// TwinCAT 3 PLC project Plc_Prog
// ProgramVersion: 3.1.4024.0
// libraries:
//   CPNTeck - OSCAT BASIC, * (CPNTeck - Automação Industrial)
//   Tc2_EtherCAT, * (Beckhoff Automation GmbH)
//   Tc2_Standard, * (Beckhoff Automation GmbH)
//   Tc2_SUPS, * (Beckhoff Automation GmbH)
//   Tc2_System, * (Beckhoff Automation GmbH)
//   Tc2_Utilities, * (Beckhoff Automation GmbH)
//   Tc3_Module, * (Beckhoff Automation GmbH)
// project tree:
//   Function Blocks/DELTA - MS300/ C2000_ANALOG_INPUTS.TcDUT (not stored), C2000_ANALOG_OUTPUTS.TcDUT (not stored), C2000_CONTROLWORD.TcDUT (not stored), C2000_DEV_CONFIG.TcDUT, C2000_DIGITAL_INPUTS.TcDUT, C2000_DIGITAL_OUTPUTS.TcDUT (not stored), C2000_DRVTOPLC_PDOS.TcDUT (not stored), C2000_PDOS.TcDUT, C2000_PLCTODRV_PDOS.TcDUT (not stored), C2000_STATUSWORD.TcDUT (not stored), E_C2000_ModeOfOperation.TcDUT, FB_DELTA_C2000_ETC.TcPOU
//   Function Blocks/IOs/Beckhoff/Common/ FB_SavePersistentData.TcPOU (not stored)
//   Function Blocks/IOs/Beckhoff/EL1809 - Digital Inputs/DataTypes/ EL1809_DEV_CONFIG.TcDUT, EL1809_HWTOPLC_PDOS.TcDUT (not stored), EL1809_PDOS.TcDUT
//   Function Blocks/IOs/Beckhoff/EL1809 - Digital Inputs/ FB_EL1809.TcPOU
//   Function Blocks/IOs/Beckhoff/EL3052 - Ai 2 x 4-20MA - 12bit/DataTypes/ EL3052_DEV_CONFIG.TcDUT (not stored), EL3052_DEV_STATUS.TcDUT (not stored), EL3052_HWTOPLC_PDOS.TcDUT (not stored), EL3052_CHANNEL.TcDUT, EL3052_PDOS.TcDUT
//   Function Blocks/IOs/Beckhoff/EL3052 - Ai 2 x 4-20MA - 12bit/ FB_EL3052.TcPOU (not stored)
//   Function Blocks/IOs/Beckhoff/EL2809 - Digital Outputs/DataTypes/ EL2809_DEV_CONFIG.TcDUT (not stored), EL2809_PDOS.TcDUT, EL2809_PLCTOHW_PDOS.TcDUT (not stored)
//   Function Blocks/IOs/Beckhoff/EL2809 - Digital Outputs/ FB_EL2809.TcPOU
//   Function Blocks/IOs/Beckhoff/EL3152 - Ai 2 x 4-20MA - 16bit/DataTypes/ EL3152_CHANNEL.TcDUT (not stored), EL3152_DEV_CONFIG.TcDUT (not stored), EL3152_DEV_STATUS.TcDUT (not stored), EL3152_HWTOPLC_PDOS.TcDUT, EL3152_PDOS.TcDUT (not stored)
//   Function Blocks/IOs/Beckhoff/EL3152 - Ai 2 x 4-20MA - 16bit/ FB_EL3152.TcPOU
//   Function Blocks/IOs/Beckhoff/EL3154 - Ai 4 x 4-20MA - 16bit/DataTypes/ EL3154_CHANNEL.TcDUT, EL3154_DEV_CONFIG.TcDUT (not stored), EL3154_DEV_STATUS.TcDUT (not stored), EL3154_HWTOPLC_PDOS.TcDUT, EL3154_PDOS.TcDUT (not stored)
//   Function Blocks/IOs/Beckhoff/EL3154 - Ai 4 x 4-20MA - 16bit/ FB_EL3154.TcPOU (not stored)
//   Function Blocks/IOs/Beckhoff/EL3204 - Ai 4 x PT100 %28RTD%29/DataTypes/ EL3204_DEV_CONFIG.TcDUT (not stored), EL3204_CHANNEL.TcDUT (not stored), EL3204_DEV_STATUS.TcDUT (not stored), EL3204_HWTOPLC_PDOS.TcDUT (not stored), EL3204_PDOS.TcDUT (not stored)
//   Function Blocks/IOs/Beckhoff/EL3204 - Ai 4 x PT100 %28RTD%29/ FB_EL3204.TcPOU (not stored)
//   Function Blocks/IOs/Beckhoff/EL4024 - AQ 4 x 4-20MA/DataTypes/ EL4024_DEV_CONFIG.TcDUT (not stored), EL4024_HWTOPLC_PDOS.TcDUT (not stored), EL4024_PDOS.TcDUT (not stored)
//   Function Blocks/IOs/Beckhoff/EL4024 - AQ 4 x 4-20MA/ FB_EL4024.TcPOU (not stored)
//   Function Blocks/IOs/Beckhoff/EL6910 - TwinSAFE PLC/ EL6910_ESTOP.TcDUT (not stored), EL6910_ESTOP_DIGNOSTICS.TcDUT (not stored), EL6910_ESTOP_STATUS.TcDUT, EL6910_HWTOPLC_PDOS.TcDUT (not stored), EL6910_PDOS.TcDUT, EL6910_PLCTOHW_PDOS.TcDUT, FB_EL6910.TcPOU (not stored)
//   Function Blocks/PaperMachine/Auxiliary/ FB_FormingBoardDriveControl.TcPOU, FB_FormingBoardRollUpDown.TcPOU, FB_FormingBoardWireStretchControl.TcPOU (not stored), FB_Gen_SRamp.TcPOU (not stored), FB_HeadboxLipsPWMControl.TcPOU (not stored), FB_LevelControl.TcPOU, FB_LevelControl_V2.TcPOU (not stored), FB_MixPumpControl.TcPOU, FB_MixPumpControl_V1.TcPOU, FB_PaperMachine.TcPOU, FB_PressureControl.TcPOU (not stored), FB_PressureControl_V1.TcPOU, FB_VfdProcessControler.TcPOU, FB_ValveProcessControler.TcPOU, FB_SimpleMotorStart.TcPOU, FB_SimpleMotorStart_V2.TcPOU, FB_SimpleMotorStart_V3.TcPOU, FB_SoftstarterSimple.TcPOU (not stored), FB_SoftstarterWithBypass.TcPOU, FB_SoftstarterWithBypass_V1.TcPOU, FB_SpeedDroopControl.TcPOU, FB_SpeedDroopControl_1.TcPOU, FB_WirePitControl.TcPOU, FB_WirePitControl_1.TcPOU (not stored)
//   Function Blocks/PaperMachine/DataTypes/ PaperMachine_TypeHmiConfig.TcDUT, PaperMachine_TypeHmiCommands.TcDUT, PaperMachine_TypeHmiStatus.TcDUT, PaperMachine_TypeHmiAlarms.TcDUT
//   Function Blocks/PaperMachine/DriveControl/ FB_DryingSectionDriveControl_V1.TcPOU (not stored), FB_DryingSectionDriveControl_V2.TcPOU (not stored), FB_DryingSectionDriveControl_V3.TcPOU, FB_FormingBoardControl_V3.TcPOU, FB_PressSectionDriveControl_V2_bak.TcPOU, FB_WinderDriveControl_V1.TcPOU, FB_DryingSectionLubrificationControl_V1.TcPOU, FB_DryingSectionPressureControl.TcPOU (not stored), FB_FormingBoardControl_V1.TcPOU, FB_PressSectionDriveControl_V1.TcPOU (not stored), FB_PressSectionDriveControl_V2.TcPOU
//   Function Blocks/PaperMachine/ FB_AlarmControl.TcPOU, FB_GroupDisplayFilters_V1.TcPOU, FB_GroupDriveControl_V1.TcPOU (not stored), FB_GroupSpeedControl_V1.TcPOU, FB_FormingBoardSpeedControl.TcPOU, FB_DryingSecSpeedControl.TcPOU, FB_WinderSpeedControl.TcPOU, FB_GroupTorqueTrimControl_V1.TcPOU, FB_GroupTorqueTrimControl_V2.TcPOU
//   Function Blocks/Rewinder/DataTypes/ RewinderConfig_TypeStruct.TcDUT (not stored), Rewinder_TypePressRoll.TcDUT, Rewinder_TypeBrakeControl.TcDUT
//   Function Blocks/Rewinder/ FB_RewinderControl_V1.TcPOU (not stored)
//   GVLs/ GVL_Hw.TcGVL (not stored)
//   / PlcTask.TcTTO
//   POUs/Implicit Checks/ CheckBounds.TcPOU (not stored), CheckDivDInt.TcPOU, CheckDivLInt.TcPOU, CheckDivLReal.TcPOU (not stored), CheckDivReal.TcPOU (not stored), CheckLRangeSigned.TcPOU (not stored), CheckLRangeUnsigned.TcPOU (not stored), CheckPointer.TcPOU (not stored), CheckRangeSigned.TcPOU (not stored), CheckRangeUnsigned.TcPOU
//   POUs/ MAIN.TcPOU
// real-time tasks:
//   TASK PlcTask: cycle T#5ms, priority 20, ADS port 350
// I/O:
//   DEVICE ETH, AmsNetId 192.168.100.1.3.1
//     +P5=050-BC1 - PLC Cabinet [EK1100 EtherCAT Coupler (2A E-Bus)]
//       +P5=050-DI1 (EL1809) [EL1809 16Ch. Dig. Input 24V, 3ms]
//       +P5=050-DI2 (EL1809) [EL1809 16Ch. Dig. Input 24V, 3ms]
//       +P5=050-DI3 (EL1809) [EL1809 16Ch. Dig. Input 24V, 3ms]
//       +P5=050-DO1 (EL2809) [EL2809 16Ch. Dig. Output 24V, 0.5A]
//       +P5=050-DO2 (EL2809) [EL2809 16Ch. Dig. Output 24V, 0.5A]
//       +P5=050-DO3 (EL2809) [EL2809 16Ch. Dig. Output 24V, 0.5A]
//       +P5=050-SP1 (EL6910) [EL6910, TwinSAFE PLC]
//       +P5=050-SI1 (EL1918) [EL1918, 8Ch. Safety Input 24V, TwinSAFE]
//         modules: Module 1 (FSOE), Module 2 (FSLOGIC)
//       +P5=050-SO1 (EL2904) [EL2904, 4 Ch. Safety Output 24V, 0.5A, TwinSAFE]
//         modules: Module 1 (FSOES), Module 2 (DO)
//       +P5=050-SO2 (EL2904) [EL2904, 4 Ch. Safety Output 24V, 0.5A, TwinSAFE]
//         modules: Module 1 (FSOES), Module 2 (DO)
//       +P5=050-BC2 [EL6601 1 Port Switch (Ethernet, CoE)]
//       +P5=050-BC3 [EL6601 1 Port Switch (Ethernet, CoE)]
//       +P5=050-BE1 [EL9011 End Terminal]
//     +P5=050-BC2 - PLC Cabinet [EK1100 EtherCAT Coupler (2A E-Bus)]
//       +P5=050-AI (EL3052) [EL3052 2Ch. Ana. Input 4-20mA]
//       +P5=050-AI2 (EL3152) [EL3152 2Ch. Ana Input 4-20mA]
//       +P5=050-AI3 (EL3052) [EL3052 2Ch. Ana. Input 4-20mA]
//       +P5=050-AI4 (EL3052) [EL3052 2Ch. Ana. Input 4-20mA]
//       +P5=050-BE2 [EL9011 End Terminal]
//     +P4=300-UG1 - Mix Pump [Delta CH2000 EtherCAT(CoE)]
//     +P3=300-UG1 - WirePit Pump [Delta CH2000 EtherCAT(CoE)]
//     +P3=100-UG1 - SuctionRoll [Delta CH2000 EtherCAT(CoE)]
//     +P3=100-UG1 - CouchPit [Delta CH2000 EtherCAT(CoE)]
//     +P3=100-UG2 - Stock pump [Delta CH2000 EtherCAT(CoE)]
//     +P2=100-UG1 - Drive Roll [Delta CH2000 EtherCAT(CoE)]
//     +P9=050-BC1 - Vaccum PLC Cabinet [EK1100 EtherCAT Coupler (2A E-Bus)]
//       +P9=050-DI1 (EL1809) [EL1809 16Ch. Dig. Input 24V, 3ms]
//       +P9=050-DI2 (EL1809) [EL1809 16Ch. Dig. Input 24V, 3ms]
//       +P9=050-DI3 (EL1809) [EL1809 16Ch. Dig. Input 24V, 3ms]
//       +P9=050-DO1 (EL2809) [EL2809 16Ch. Dig. Output 24V, 0.5A]
//       +P9=050-DO2 (EL2809) [EL2809 16Ch. Dig. Output 24V, 0.5A]
//       +P9=050-DO3 (EL2809) [EL2809 16Ch. Dig. Output 24V, 0.5A]
//       +P9=050-AI1 (EL3054) [EL3054 4Ch. Ana. Input 4-20mA]
//       Term 101 (EL3052) [EL3052 2Ch. Ana. Input 4-20mA]
//       Term 102 (EL4004) [EL4004 4Ch. Ana. Output 0-10V, 12bit]
//       Term 151 (EL9011) [EL9011 End Terminal]
//       +P9=050-BE1 [EL9011 End Terminal]
//     +P10=050-BC1 - Press / Dryer PLC Cabinet [EK1100 EtherCAT Coupler (2A E-Bus)]
//       +P10=050-DI1 (EL1809) [EL1809 16Ch. Dig. Input 24V, 3ms]
//       +P10=050-DI2 (EL1809) [EL1809 16Ch. Dig. Input 24V, 3ms]
//       +P10=050-DI3 (EL1809) [EL1809 16Ch. Dig. Input 24V, 3ms]
//       +P10=050-DI4 (EL1809) [EL1809 16Ch. Dig. Input 24V, 3ms]
//       +P10=050-DI5 (EL1809) [EL1809 16Ch. Dig. Input 24V, 3ms]
//       +P10=050-DI6 (EL1809) [EL1809 16Ch. Dig. Input 24V, 3ms]
//       +P10=050-DI7 (EL1809) [EL1809 16Ch. Dig. Input 24V, 3ms]
//       +P10=050-DI8 (EL1809) [EL1809 16Ch. Dig. Input 24V, 3ms]
//       +P10=050-DO1 (EL2809) [EL2809 16Ch. Dig. Output 24V, 0.5A]
//       +P10=050-DO2 (EL2809) [EL2809 16Ch. Dig. Output 24V, 0.5A]
//       +P10=050-DO3 (EL2809) [EL2809 16Ch. Dig. Output 24V, 0.5A]
//       +P10=050-DO4 (EL2809) [EL2809 16Ch. Dig. Output 24V, 0.5A]
//       +P10=050-SI1 (EL1918) [EL1918, 8Ch. Safety Input 24V, TwinSAFE]
//         modules: Module 1 (FSOE), Module 2 (FSLOGIC)
//       +P10=050-SO1 (EL2904) [EL2904, 4 Ch. Safety Output 24V, 0.5A, TwinSAFE]
//         modules: Module 1 (FSOES), Module 2 (DO)
//       +P10=050-BE1 [EL9011 End Terminal]
//     +P10=050-BC2 - Press / Dryer PLC Cabinet [EK1100 EtherCAT Coupler (2A E-Bus)]
//       +P10=050-AI1 (EL3054) [EL3054 4Ch. Ana. Input 4-20mA]
//       +P10=050-AI2 (EL3204) [EL3204 4Ch. Ana. Input PT100 (RTD)]
//       +P10=050-AO1(EL4024) [EL4024 4Ch. Ana. Output 4-20mA, 12bit]
//       +P10=050-BE2 [EL9011 End Terminal]
//     +P11=400-UG1 - Second Press [Delta C2000Plus EtherCAT(CoE)]
//     +P12=400-UG1 - First Press [Delta C2000Plus EtherCAT(CoE)]
//     +P13=500-UG1 - Dryer Section GR1 - Upper GR1 Slave [Delta C2000Plus EtherCAT(CoE)]
//     +P12=500-UG2 - Dryer Section GR1 - Lower GR1 Master [Delta C2000Plus EtherCAT(CoE)]
//     +P12=500-UG3 - Dryer Section GR1 - Upper Master [Delta CH2000 EtherCAT(CoE)]
//     +P12=501-UG1 - Dryer Section  GR2 - Lower Slave [Delta C2000Plus EtherCAT(CoE)]
//     +P12=501-UG2 - Dryer Section GR2 - Upper Slave [Delta CH2000 EtherCAT(CoE)]
//     +P12=501-UG3 - Dryer Section GR2 - Lower Master [Delta C2000Plus EtherCAT(CoE)]
//     +P13=501-UG1 - Dryer Section GR2 - Upper Master [Delta CH2000 EtherCAT(CoE)]
//     +P13=502-UG2 - Dryer Section GR3 - Lower Slave [Delta C2000Plus EtherCAT(CoE)]
//     +P13=502-UG2 - Dryer Section GR3 - Upper Slave [Delta C2000Plus EtherCAT(CoE)]
//     +P13=502-UG3 - Dryer Section GR3 - Lower Master [Delta C2000Plus EtherCAT(CoE)]
//     +P13=502-UG4 - Dryer Section GR3 - Upper Master [Delta C2000Plus EtherCAT(CoE)]
//     +P14=600-UG1 - Winder [Delta C2000Plus EtherCAT(CoE)]
//     +CP2=050-BC1 - Winder command panel [EK1100 EtherCAT Coupler (2A E-Bus)]
//       +CP2=050-SI1 (EL1918) [EL1918, 8Ch. Safety Input 24V, TwinSAFE]
//         modules: Module 1 (FSOE), Module 2 (FSLOGIC)
//       +CP2=050-DI1 (EL1809) [EL1809 16Ch. Dig. Input 24V, 3ms]
//       +CP2=050-DO1 (EL2809 [EL2809 16Ch. Dig. Output 24V, 0.5A]
//       +CP2=050-AO1 (EL4024) [EL4024 4Ch. Ana. Output 4-20mA, 12bit]
//       +CP2=050-BE1 (EL4024) [EL9011 End Terminal]
// variable links:
//   ETH <-> ETH/+CP2=050-BC1 - Winder command panel/+CP2=050-SI1 (EL1918)
//     +P5=050-BC1 - PLC Cabinet/+P5=050-SP1 (EL6910)/ConnectionInputs/TwinSafeGroup1.+CP2=050-SI1 (EL1918) - Module 1 (FSOE)_9 TxPDO <-> Module 1 (FSOE)/FSoE Outputs/FSOE
//     +P5=050-BC1 - PLC Cabinet/+P5=050-SP1 (EL6910)/ConnectionOutputs/TwinSafeGroup1.+CP2=050-SI1 (EL1918) - Module 1 (FSOE)_9 RxPDO <-> Module 1 (FSOE)/FSoE Inputs/FSOE
//   ETH <-> ETH/+P10=050-BC1 - Press / Dryer PLC Cabinet/+P10=050-SI1 (EL1918)
//     +P5=050-BC1 - PLC Cabinet/+P5=050-SP1 (EL6910)/ConnectionInputs/TwinSafeGroup1.+P10=050-SI1 (EL1918) - Module 1 (FSOE)_7 TxPDO <-> Module 1 (FSOE)/FSoE Outputs/FSOE
//   ETH <-> ETH/+P10=050-BC1 - Press / Dryer PLC Cabinet/+P10=050-SO1 (EL2904)
//     +P5=050-BC1 - PLC Cabinet/+P5=050-SP1 (EL6910)/ConnectionInputs/TwinSafeGroup1.+P10=050-SO1 (EL2904) - Module 1 (FSOES)_8 TxPDO <-> Module 1 (FSOES)/RxPDO/FSOE
//     +P5=050-BC1 - PLC Cabinet/+P5=050-SP1 (EL6910)/ConnectionOutputs/TwinSafeGroup1.+P10=050-SO1 (EL2904) - Module 1 (FSOES)_8 RxPDO <-> Module 1 (FSOES)/TxPDO/FSOE
//   ETH <-> ETH/+P5=050-BC1 - PLC Cabinet/+P5=050-SI1 (EL1918)
//     +P5=050-BC1 - PLC Cabinet/+P5=050-SP1 (EL6910)/ConnectionInputs/TwinSafeGroup1.Term 9 (EL1918) - Module 1 (FSOE)_3 TxPDO <-> Module 1 (FSOE)/FSoE Outputs/FSOE
//   ETH <-> ETH/+P5=050-BC1 - PLC Cabinet/+P5=050-SP1 (EL6910)
//     +P10=050-BC1 - Press / Dryer PLC Cabinet/+P10=050-SI1 (EL1918)/Module 1 (FSOE)/FSoE Inputs/FSOE <-> ConnectionOutputs/TwinSafeGroup1.+P10=050-SI1 (EL1918) - Module 1 (FSOE)_7 RxPDO
//     +P5=050-BC1 - PLC Cabinet/+P5=050-SI1 (EL1918)/Module 1 (FSOE)/FSoE Inputs/FSOE <-> ConnectionOutputs/TwinSafeGroup1.Term 9 (EL1918) - Module 1 (FSOE)_3 RxPDO
//     +P5=050-BC1 - PLC Cabinet/+P5=050-SO1 (EL2904)/Module 1 (FSOES)/RxPDO/FSOE <-> ConnectionInputs/TwinSafeGroup1.Term 10 (EL2904) - Module 1 (FSOES)_4 TxPDO
//     +P5=050-BC1 - PLC Cabinet/+P5=050-SO2 (EL2904)/Module 1 (FSOES)/RxPDO/FSOE <-> ConnectionInputs/TwinSafeGroup1.Term 11 (EL2904) - Module 1 (FSOES)_5 TxPDO
//     +P5=050-BC1 - PLC Cabinet/+P5=050-SO1 (EL2904)/Module 1 (FSOES)/TxPDO/FSOE <-> ConnectionOutputs/TwinSafeGroup1.Term 10 (EL2904) - Module 1 (FSOES)_4 RxPDO
//     +P5=050-BC1 - PLC Cabinet/+P5=050-SO2 (EL2904)/Module 1 (FSOES)/TxPDO/FSOE <-> ConnectionOutputs/TwinSafeGroup1.Term 11 (EL2904) - Module 1 (FSOES)_5 RxPDO
//   Plc_Prog/Plc_Prog Instance <-> ETH/+CP2=050-BC1 - Winder command panel/+CP2=050-AO1 (EL4024)
//     PlcTask Outputs/.CP1_050_AO1.PDOS.HwToPLC.Channel1 <-> AO Outputs Channel 1/Analog output
//     PlcTask Outputs/.CP1_050_AO1.PDOS.HwToPLC.Channel2 <-> AO Outputs Channel 2/Analog output
//     PlcTask Outputs/.CP1_050_AO1.PDOS.HwToPLC.Channel3 <-> AO Outputs Channel 3/Analog output
//     PlcTask Outputs/.CP1_050_AO1.PDOS.HwToPLC.Channel4 <-> AO Outputs Channel 4/Analog output
//   Plc_Prog/Plc_Prog Instance <-> ETH/+CP2=050-BC1 - Winder command panel/+CP2=050-DI1 (EL1809)
//     PlcTask Inputs/.CP1_050_DI1.PDOS.digitalInput_01 <-> Channel 1/Input
//     PlcTask Inputs/.CP1_050_DI1.PDOS.digitalInput_02 <-> Channel 2/Input
//     PlcTask Inputs/.CP1_050_DI1.PDOS.digitalInput_03 <-> Channel 3/Input
//     PlcTask Inputs/.CP1_050_DI1.PDOS.digitalInput_04 <-> Channel 4/Input
//     PlcTask Inputs/.CP1_050_DI1.PDOS.digitalInput_05 <-> Channel 5/Input
//     PlcTask Inputs/.CP1_050_DI1.PDOS.digitalInput_06 <-> Channel 6/Input
//     PlcTask Inputs/.CP1_050_DI1.PDOS.digitalInput_07 <-> Channel 7/Input
//     PlcTask Inputs/.CP1_050_DI1.PDOS.digitalInput_08 <-> Channel 8/Input
//     PlcTask Inputs/.CP1_050_DI1.PDOS.digitalInput_09 <-> Channel 9/Input
//     PlcTask Inputs/.CP1_050_DI1.PDOS.digitalInput_10 <-> Channel 10/Input
//     PlcTask Inputs/.CP1_050_DI1.PDOS.digitalInput_11 <-> Channel 11/Input
//     PlcTask Inputs/.CP1_050_DI1.PDOS.digitalInput_12 <-> Channel 12/Input
//     PlcTask Inputs/.CP1_050_DI1.PDOS.digitalInput_13 <-> Channel 13/Input
//     PlcTask Inputs/.CP1_050_DI1.PDOS.digitalInput_14 <-> Channel 14/Input
//     PlcTask Inputs/.CP1_050_DI1.PDOS.digitalInput_15 <-> Channel 15/Input
//     PlcTask Inputs/.CP1_050_DI1.PDOS.digitalInput_16 <-> Channel 16/Input
//   Plc_Prog/Plc_Prog Instance <-> ETH/+CP2=050-BC1 - Winder command panel/+CP2=050-DO1 (EL2809
//     PlcTask Outputs/.CP1_050_DO1.PDOS.PlcToHw.digitalOutput_01 <-> Channel 1/Output
//     PlcTask Outputs/.CP1_050_DO1.PDOS.PlcToHw.digitalOutput_02 <-> Channel 2/Output
//     PlcTask Outputs/.CP1_050_DO1.PDOS.PlcToHw.digitalOutput_03 <-> Channel 3/Output
//     PlcTask Outputs/.CP1_050_DO1.PDOS.PlcToHw.digitalOutput_04 <-> Channel 4/Output
//     PlcTask Outputs/.CP1_050_DO1.PDOS.PlcToHw.digitalOutput_05 <-> Channel 5/Output
//     PlcTask Outputs/.CP1_050_DO1.PDOS.PlcToHw.digitalOutput_06 <-> Channel 6/Output
//     PlcTask Outputs/.CP1_050_DO1.PDOS.PlcToHw.digitalOutput_07 <-> Channel 7/Output
//     PlcTask Outputs/.CP1_050_DO1.PDOS.PlcToHw.digitalOutput_08 <-> Channel 8/Output
//     PlcTask Outputs/.CP1_050_DO1.PDOS.PlcToHw.digitalOutput_09 <-> Channel 9/Output
//     PlcTask Outputs/.CP1_050_DO1.PDOS.PlcToHw.digitalOutput_10 <-> Channel 10/Output
//     PlcTask Outputs/.CP1_050_DO1.PDOS.PlcToHw.digitalOutput_11 <-> Channel 11/Output
//     PlcTask Outputs/.CP1_050_DO1.PDOS.PlcToHw.digitalOutput_12 <-> Channel 12/Output
//     PlcTask Outputs/.CP1_050_DO1.PDOS.PlcToHw.digitalOutput_13 <-> Channel 13/Output
//     PlcTask Outputs/.CP1_050_DO1.PDOS.PlcToHw.digitalOutput_14 <-> Channel 14/Output
//     PlcTask Outputs/.CP1_050_DO1.PDOS.PlcToHw.digitalOutput_15 <-> Channel 15/Output
//     PlcTask Outputs/.CP1_050_DO1.PDOS.PlcToHw.digitalOutput_16 <-> Channel 16/Output
//   Plc_Prog/Plc_Prog Instance <-> ETH/+P10=050-BC1 - Press / Dryer PLC Cabinet/+P10=050-DI1 (EL1809)
//     PlcTask Inputs/.P10_050_DI1.PDOS.digitalInput_01 <-> Channel 1/Input
//     PlcTask Inputs/.P10_050_DI1.PDOS.digitalInput_02 <-> Channel 2/Input
//     PlcTask Inputs/.P10_050_DI1.PDOS.digitalInput_03 <-> Channel 3/Input
//     PlcTask Inputs/.P10_050_DI1.PDOS.digitalInput_04 <-> Channel 4/Input
//     PlcTask Inputs/.P10_050_DI1.PDOS.digitalInput_05 <-> Channel 5/Input
//     PlcTask Inputs/.P10_050_DI1.PDOS.digitalInput_06 <-> Channel 6/Input
//     PlcTask Inputs/.P10_050_DI1.PDOS.digitalInput_07 <-> Channel 7/Input
//     PlcTask Inputs/.P10_050_DI1.PDOS.digitalInput_08 <-> Channel 8/Input
//     PlcTask Inputs/.P10_050_DI1.PDOS.digitalInput_09 <-> Channel 9/Input
//     PlcTask Inputs/.P10_050_DI1.PDOS.digitalInput_10 <-> Channel 10/Input
//     PlcTask Inputs/.P10_050_DI1.PDOS.digitalInput_11 <-> Channel 11/Input
//     PlcTask Inputs/.P10_050_DI1.PDOS.digitalInput_12 <-> Channel 12/Input
//     PlcTask Inputs/.P10_050_DI1.PDOS.digitalInput_13 <-> Channel 13/Input
//     PlcTask Inputs/.P10_050_DI1.PDOS.digitalInput_14 <-> Channel 14/Input
//     PlcTask Inputs/.P10_050_DI1.PDOS.digitalInput_15 <-> Channel 15/Input
//     PlcTask Inputs/.P10_050_DI1.PDOS.digitalInput_16 <-> Channel 16/Input
//   Plc_Prog/Plc_Prog Instance <-> ETH/+P10=050-BC1 - Press / Dryer PLC Cabinet/+P10=050-DI2 (EL1809)
//     PlcTask Inputs/.P10_050_DI2.PDOS.digitalInput_01 <-> Channel 1/Input
//     PlcTask Inputs/.P10_050_DI2.PDOS.digitalInput_02 <-> Channel 2/Input
//     PlcTask Inputs/.P10_050_DI2.PDOS.digitalInput_03 <-> Channel 3/Input
//     PlcTask Inputs/.P10_050_DI2.PDOS.digitalInput_04 <-> Channel 4/Input
//     PlcTask Inputs/.P10_050_DI2.PDOS.digitalInput_05 <-> Channel 5/Input
//     PlcTask Inputs/.P10_050_DI2.PDOS.digitalInput_06 <-> Channel 6/Input
//     PlcTask Inputs/.P10_050_DI2.PDOS.digitalInput_07 <-> Channel 7/Input
//     PlcTask Inputs/.P10_050_DI2.PDOS.digitalInput_08 <-> Channel 8/Input
//     PlcTask Inputs/.P10_050_DI2.PDOS.digitalInput_09 <-> Channel 9/Input
//     PlcTask Inputs/.P10_050_DI2.PDOS.digitalInput_10 <-> Channel 10/Input
//     PlcTask Inputs/.P10_050_DI2.PDOS.digitalInput_12 <-> Channel 12/Input
//     PlcTask Inputs/.P10_050_DI2.PDOS.digitalInput_13 <-> Channel 13/Input
//     PlcTask Inputs/.P10_050_DI2.PDOS.digitalInput_14 <-> Channel 14/Input
//     PlcTask Inputs/.P10_050_DI2.PDOS.digitalInput_15 <-> Channel 15/Input
//     PlcTask Inputs/.P10_050_DI2.PDOS.digitalInput_16 <-> Channel 16/Input
//     PlcTask Inputs/.P10_050_DI2.PDOS.digitalInput_11 <-> Channel 11/.P10_050_DI2.PDOS.digitalInput_11
//   Plc_Prog/Plc_Prog Instance <-> ETH/+P10=050-BC1 - Press / Dryer PLC Cabinet/+P10=050-DI3 (EL1809)
//     PlcTask Inputs/.P10_050_DI3.PDOS.digitalInput_01 <-> Channel 1/Input
//     PlcTask Inputs/.P10_050_DI3.PDOS.digitalInput_02 <-> Channel 2/Input
//     PlcTask Inputs/.P10_050_DI3.PDOS.digitalInput_03 <-> Channel 3/Input
//     PlcTask Inputs/.P10_050_DI3.PDOS.digitalInput_04 <-> Channel 4/Input
//     PlcTask Inputs/.P10_050_DI3.PDOS.digitalInput_05 <-> Channel 5/Input
//     PlcTask Inputs/.P10_050_DI3.PDOS.digitalInput_06 <-> Channel 6/Input
//     PlcTask Inputs/.P10_050_DI3.PDOS.digitalInput_07 <-> Channel 7/Input
//     PlcTask Inputs/.P10_050_DI3.PDOS.digitalInput_08 <-> Channel 8/Input
//     PlcTask Inputs/.P10_050_DI3.PDOS.digitalInput_09 <-> Channel 9/Input
//     PlcTask Inputs/.P10_050_DI3.PDOS.digitalInput_10 <-> Channel 10/Input
//     PlcTask Inputs/.P10_050_DI3.PDOS.digitalInput_11 <-> Channel 11/Input
//     PlcTask Inputs/.P10_050_DI3.PDOS.digitalInput_12 <-> Channel 12/Input
//     PlcTask Inputs/.P10_050_DI3.PDOS.digitalInput_13 <-> Channel 13/Input
//     PlcTask Inputs/.P10_050_DI3.PDOS.digitalInput_14 <-> Channel 14/Input
//     PlcTask Inputs/.P10_050_DI3.PDOS.digitalInput_15 <-> Channel 15/Input
//     PlcTask Inputs/.P10_050_DI3.PDOS.digitalInput_16 <-> Channel 16/Input
//   Plc_Prog/Plc_Prog Instance <-> ETH/+P10=050-BC1 - Press / Dryer PLC Cabinet/+P10=050-DI4 (EL1809)
//     PlcTask Inputs/.P10_050_DI4.PDOS.digitalInput_01 <-> Channel 1/Input
//     PlcTask Inputs/.P10_050_DI4.PDOS.digitalInput_02 <-> Channel 2/Input
//     PlcTask Inputs/.P10_050_DI4.PDOS.digitalInput_03 <-> Channel 3/Input
//     PlcTask Inputs/.P10_050_DI4.PDOS.digitalInput_04 <-> Channel 4/Input
//     PlcTask Inputs/.P10_050_DI4.PDOS.digitalInput_05 <-> Channel 5/Input
//     PlcTask Inputs/.P10_050_DI4.PDOS.digitalInput_06 <-> Channel 6/Input
//     PlcTask Inputs/.P10_050_DI4.PDOS.digitalInput_07 <-> Channel 7/Input
//     PlcTask Inputs/.P10_050_DI4.PDOS.digitalInput_08 <-> Channel 8/Input
//     PlcTask Inputs/.P10_050_DI4.PDOS.digitalInput_09 <-> Channel 9/Input
//     PlcTask Inputs/.P10_050_DI4.PDOS.digitalInput_10 <-> Channel 10/Input
//     PlcTask Inputs/.P10_050_DI4.PDOS.digitalInput_11 <-> Channel 11/Input
//     PlcTask Inputs/.P10_050_DI4.PDOS.digitalInput_12 <-> Channel 12/Input
//     PlcTask Inputs/.P10_050_DI4.PDOS.digitalInput_13 <-> Channel 13/Input
//     PlcTask Inputs/.P10_050_DI4.PDOS.digitalInput_14 <-> Channel 14/Input
//     PlcTask Inputs/.P10_050_DI4.PDOS.digitalInput_15 <-> Channel 15/Input
//     PlcTask Inputs/.P10_050_DI4.PDOS.digitalInput_16 <-> Channel 16/Input
//   Plc_Prog/Plc_Prog Instance <-> ETH/+P10=050-BC1 - Press / Dryer PLC Cabinet/+P10=050-DI5 (EL1809)
//     PlcTask Inputs/.P10_050_DI5.PDOS.digitalInput_01 <-> Channel 1/Input
//     PlcTask Inputs/.P10_050_DI5.PDOS.digitalInput_02 <-> Channel 2/Input
//     PlcTask Inputs/.P10_050_DI5.PDOS.digitalInput_03 <-> Channel 3/Input
//     PlcTask Inputs/.P10_050_DI5.PDOS.digitalInput_04 <-> Channel 4/Input
//     PlcTask Inputs/.P10_050_DI5.PDOS.digitalInput_05 <-> Channel 5/Input
//     PlcTask Inputs/.P10_050_DI5.PDOS.digitalInput_06 <-> Channel 6/Input
//     PlcTask Inputs/.P10_050_DI5.PDOS.digitalInput_07 <-> Channel 7/Input
//     PlcTask Inputs/.P10_050_DI5.PDOS.digitalInput_08 <-> Channel 8/Input
//     PlcTask Inputs/.P10_050_DI5.PDOS.digitalInput_09 <-> Channel 9/Input
//     PlcTask Inputs/.P10_050_DI5.PDOS.digitalInput_10 <-> Channel 10/Input
//     PlcTask Inputs/.P10_050_DI5.PDOS.digitalInput_11 <-> Channel 11/Input
//     PlcTask Inputs/.P10_050_DI5.PDOS.digitalInput_12 <-> Channel 12/Input
//     PlcTask Inputs/.P10_050_DI5.PDOS.digitalInput_13 <-> Channel 13/Input
//     PlcTask Inputs/.P10_050_DI5.PDOS.digitalInput_14 <-> Channel 14/Input
//     PlcTask Inputs/.P10_050_DI5.PDOS.digitalInput_15 <-> Channel 15/Input
//     PlcTask Inputs/.P10_050_DI5.PDOS.digitalInput_16 <-> Channel 16/Input
//   Plc_Prog/Plc_Prog Instance <-> ETH/+P10=050-BC1 - Press / Dryer PLC Cabinet/+P10=050-DI6 (EL1809)
//     PlcTask Inputs/.P10_050_DI6.PDOS.digitalInput_01 <-> Channel 1/Input
//     PlcTask Inputs/.P10_050_DI6.PDOS.digitalInput_02 <-> Channel 2/Input
//     PlcTask Inputs/.P10_050_DI6.PDOS.digitalInput_03 <-> Channel 3/Input
//     PlcTask Inputs/.P10_050_DI6.PDOS.digitalInput_04 <-> Channel 4/Input
//     PlcTask Inputs/.P10_050_DI6.PDOS.digitalInput_05 <-> Channel 5/Input
//     PlcTask Inputs/.P10_050_DI6.PDOS.digitalInput_06 <-> Channel 6/Input
//     PlcTask Inputs/.P10_050_DI6.PDOS.digitalInput_07 <-> Channel 7/Input
//     PlcTask Inputs/.P10_050_DI6.PDOS.digitalInput_08 <-> Channel 8/Input
//     PlcTask Inputs/.P10_050_DI6.PDOS.digitalInput_09 <-> Channel 9/Input
//     PlcTask Inputs/.P10_050_DI6.PDOS.digitalInput_10 <-> Channel 10/Input
//     PlcTask Inputs/.P10_050_DI6.PDOS.digitalInput_11 <-> Channel 11/Input
//     PlcTask Inputs/.P10_050_DI6.PDOS.digitalInput_12 <-> Channel 12/Input
//     PlcTask Inputs/.P10_050_DI6.PDOS.digitalInput_13 <-> Channel 13/Input
//     PlcTask Inputs/.P10_050_DI6.PDOS.digitalInput_14 <-> Channel 14/Input
//     PlcTask Inputs/.P10_050_DI6.PDOS.digitalInput_15 <-> Channel 15/Input
//     PlcTask Inputs/.P10_050_DI6.PDOS.digitalInput_16 <-> Channel 16/Input
//   Plc_Prog/Plc_Prog Instance <-> ETH/+P10=050-BC1 - Press / Dryer PLC Cabinet/+P10=050-DI7 (EL1809)
//     PlcTask Inputs/.P10_050_DI7.PDOS.digitalInput_01 <-> Channel 1/Input
//     PlcTask Inputs/.P10_050_DI7.PDOS.digitalInput_02 <-> Channel 2/Input
//     PlcTask Inputs/.P10_050_DI7.PDOS.digitalInput_03 <-> Channel 3/Input
//     PlcTask Inputs/.P10_050_DI7.PDOS.digitalInput_04 <-> Channel 4/Input
//     PlcTask Inputs/.P10_050_DI7.PDOS.digitalInput_05 <-> Channel 5/Input
//     PlcTask Inputs/.P10_050_DI7.PDOS.digitalInput_06 <-> Channel 6/Input
//     PlcTask Inputs/.P10_050_DI7.PDOS.digitalInput_07 <-> Channel 7/Input
//     PlcTask Inputs/.P10_050_DI7.PDOS.digitalInput_08 <-> Channel 8/Input
//     PlcTask Inputs/.P10_050_DI7.PDOS.digitalInput_09 <-> Channel 9/Input
//     PlcTask Inputs/.P10_050_DI7.PDOS.digitalInput_10 <-> Channel 10/Input
//     PlcTask Inputs/.P10_050_DI7.PDOS.digitalInput_11 <-> Channel 11/Input
//     PlcTask Inputs/.P10_050_DI7.PDOS.digitalInput_12 <-> Channel 12/Input
//     PlcTask Inputs/.P10_050_DI7.PDOS.digitalInput_13 <-> Channel 13/Input
//     PlcTask Inputs/.P10_050_DI7.PDOS.digitalInput_14 <-> Channel 14/Input
//     PlcTask Inputs/.P10_050_DI7.PDOS.digitalInput_15 <-> Channel 15/Input
//     PlcTask Inputs/.P10_050_DI7.PDOS.digitalInput_16 <-> Channel 16/Input
//   Plc_Prog/Plc_Prog Instance <-> ETH/+P10=050-BC1 - Press / Dryer PLC Cabinet/+P10=050-DI8 (EL1809)
//     PlcTask Inputs/.P10_050_DI8.PDOS.digitalInput_01 <-> Channel 1/Input
//     PlcTask Inputs/.P10_050_DI8.PDOS.digitalInput_02 <-> Channel 2/Input
//     PlcTask Inputs/.P10_050_DI8.PDOS.digitalInput_03 <-> Channel 3/Input
//     PlcTask Inputs/.P10_050_DI8.PDOS.digitalInput_04 <-> Channel 4/Input
//     PlcTask Inputs/.P10_050_DI8.PDOS.digitalInput_05 <-> Channel 5/Input
//     PlcTask Inputs/.P10_050_DI8.PDOS.digitalInput_06 <-> Channel 6/Input
//     PlcTask Inputs/.P10_050_DI8.PDOS.digitalInput_07 <-> Channel 7/Input
//     PlcTask Inputs/.P10_050_DI8.PDOS.digitalInput_08 <-> Channel 8/Input
//     PlcTask Inputs/.P10_050_DI8.PDOS.digitalInput_09 <-> Channel 9/Input
//     PlcTask Inputs/.P10_050_DI8.PDOS.digitalInput_10 <-> Channel 10/Input
//     PlcTask Inputs/.P10_050_DI8.PDOS.digitalInput_11 <-> Channel 11/Input
//     PlcTask Inputs/.P10_050_DI8.PDOS.digitalInput_14 <-> Channel 14/Input
//     PlcTask Inputs/.P10_050_DI8.PDOS.digitalInput_16 <-> Channel 16/Input
//     PlcTask Inputs/.P10_050_DI8.PDOS.digitalInput_12 <-> Channel 12/Pressao Alta HPU
//     PlcTask Inputs/.P10_050_DI8.PDOS.digitalInput_13 <-> Channel 13/Pressao Baixa HPU
//     PlcTask Inputs/.P10_050_DI8.PDOS.digitalInput_15 <-> Channel 15/Nivel muito baixo HPU
//   Plc_Prog/Plc_Prog Instance <-> ETH/+P10=050-BC1 - Press / Dryer PLC Cabinet/+P10=050-DO1 (EL2809)
//     PlcTask Outputs/.P10_050_DO1.PDOS.PlcToHw.digitalOutput_01 <-> Channel 1/Output
//     PlcTask Outputs/.P10_050_DO1.PDOS.PlcToHw.digitalOutput_02 <-> Channel 2/Output
//     PlcTask Outputs/.P10_050_DO1.PDOS.PlcToHw.digitalOutput_03 <-> Channel 3/Output
//     PlcTask Outputs/.P10_050_DO1.PDOS.PlcToHw.digitalOutput_04 <-> Channel 4/Output
//     PlcTask Outputs/.P10_050_DO1.PDOS.PlcToHw.digitalOutput_05 <-> Channel 5/Output
//     PlcTask Outputs/.P10_050_DO1.PDOS.PlcToHw.digitalOutput_06 <-> Channel 6/Output
//     PlcTask Outputs/.P10_050_DO1.PDOS.PlcToHw.digitalOutput_07 <-> Channel 7/Output
//     PlcTask Outputs/.P10_050_DO1.PDOS.PlcToHw.digitalOutput_08 <-> Channel 8/Output
//     PlcTask Outputs/.P10_050_DO1.PDOS.PlcToHw.digitalOutput_09 <-> Channel 9/Output
//     PlcTask Outputs/.P10_050_DO1.PDOS.PlcToHw.digitalOutput_10 <-> Channel 10/Output
//     PlcTask Outputs/.P10_050_DO1.PDOS.PlcToHw.digitalOutput_11 <-> Channel 11/Output
//     PlcTask Outputs/.P10_050_DO1.PDOS.PlcToHw.digitalOutput_12 <-> Channel 12/Output
//     PlcTask Outputs/.P10_050_DO1.PDOS.PlcToHw.digitalOutput_13 <-> Channel 13/Output
//     PlcTask Outputs/.P10_050_DO1.PDOS.PlcToHw.digitalOutput_14 <-> Channel 14/Output
//     PlcTask Outputs/.P10_050_DO1.PDOS.PlcToHw.digitalOutput_15 <-> Channel 15/Output
//     PlcTask Outputs/.P10_050_DO1.PDOS.PlcToHw.digitalOutput_16 <-> Channel 16/Output
//   Plc_Prog/Plc_Prog Instance <-> ETH/+P10=050-BC1 - Press / Dryer PLC Cabinet/+P10=050-DO2 (EL2809)
//     PlcTask Outputs/.P10_050_DO2.PDOS.PlcToHw.digitalOutput_01 <-> Channel 1/Output
//     PlcTask Outputs/.P10_050_DO2.PDOS.PlcToHw.digitalOutput_02 <-> Channel 2/Output
//     PlcTask Outputs/.P10_050_DO2.PDOS.PlcToHw.digitalOutput_03 <-> Channel 3/Output
//     PlcTask Outputs/.P10_050_DO2.PDOS.PlcToHw.digitalOutput_04 <-> Channel 4/Output
//     PlcTask Outputs/.P10_050_DO2.PDOS.PlcToHw.digitalOutput_05 <-> Channel 5/Output
//     PlcTask Outputs/.P10_050_DO2.PDOS.PlcToHw.digitalOutput_06 <-> Channel 6/Output
//     PlcTask Outputs/.P10_050_DO2.PDOS.PlcToHw.digitalOutput_07 <-> Channel 7/Output
//     PlcTask Outputs/.P10_050_DO2.PDOS.PlcToHw.digitalOutput_08 <-> Channel 8/Output
//     PlcTask Outputs/.P10_050_DO2.PDOS.PlcToHw.digitalOutput_09 <-> Channel 9/Output
//     PlcTask Outputs/.P10_050_DO2.PDOS.PlcToHw.digitalOutput_10 <-> Channel 10/Output
//     PlcTask Outputs/.P10_050_DO2.PDOS.PlcToHw.digitalOutput_11 <-> Channel 11/Output
//     PlcTask Outputs/.P10_050_DO2.PDOS.PlcToHw.digitalOutput_12 <-> Channel 12/Output
//     PlcTask Outputs/.P10_050_DO2.PDOS.PlcToHw.digitalOutput_13 <-> Channel 13/Output
//     PlcTask Outputs/.P10_050_DO2.PDOS.PlcToHw.digitalOutput_14 <-> Channel 14/Output
//     PlcTask Outputs/.P10_050_DO2.PDOS.PlcToHw.digitalOutput_15 <-> Channel 15/Output
//     PlcTask Outputs/.P10_050_DO2.PDOS.PlcToHw.digitalOutput_16 <-> Channel 16/Output
//   Plc_Prog/Plc_Prog Instance <-> ETH/+P10=050-BC1 - Press / Dryer PLC Cabinet/+P10=050-DO3 (EL2809)
//     PlcTask Outputs/.P10_050_DO3.PDOS.PlcToHw.digitalOutput_01 <-> Channel 1/Output
//     PlcTask Outputs/.P10_050_DO3.PDOS.PlcToHw.digitalOutput_02 <-> Channel 2/Output
//     PlcTask Outputs/.P10_050_DO3.PDOS.PlcToHw.digitalOutput_03 <-> Channel 3/Output
//     PlcTask Outputs/.P10_050_DO3.PDOS.PlcToHw.digitalOutput_04 <-> Channel 4/Output
//     PlcTask Outputs/.P10_050_DO3.PDOS.PlcToHw.digitalOutput_05 <-> Channel 5/Output
//     PlcTask Outputs/.P10_050_DO3.PDOS.PlcToHw.digitalOutput_06 <-> Channel 6/Output
//     PlcTask Outputs/.P10_050_DO3.PDOS.PlcToHw.digitalOutput_07 <-> Channel 7/Output
//     PlcTask Outputs/.P10_050_DO3.PDOS.PlcToHw.digitalOutput_08 <-> Channel 8/Output
//     PlcTask Outputs/.P10_050_DO3.PDOS.PlcToHw.digitalOutput_09 <-> Channel 9/Output
//     PlcTask Outputs/.P10_050_DO3.PDOS.PlcToHw.digitalOutput_10 <-> Channel 10/Output
//     PlcTask Outputs/.P10_050_DO3.PDOS.PlcToHw.digitalOutput_11 <-> Channel 11/Output
//     PlcTask Outputs/.P10_050_DO3.PDOS.PlcToHw.digitalOutput_12 <-> Channel 12/Output
//     PlcTask Outputs/.P10_050_DO3.PDOS.PlcToHw.digitalOutput_13 <-> Channel 13/Output
//     PlcTask Outputs/.P10_050_DO3.PDOS.PlcToHw.digitalOutput_14 <-> Channel 14/Output
//     PlcTask Outputs/.P10_050_DO3.PDOS.PlcToHw.digitalOutput_15 <-> Channel 15/Output
//     PlcTask Outputs/.P10_050_DO3.PDOS.PlcToHw.digitalOutput_16 <-> Channel 16/Output
//   Plc_Prog/Plc_Prog Instance <-> ETH/+P10=050-BC1 - Press / Dryer PLC Cabinet/+P10=050-DO4 (EL2809)
//     PlcTask Outputs/.P10_050_DO4.PDOS.PlcToHw.digitalOutput_01 <-> Channel 1/Output
//     PlcTask Outputs/.P10_050_DO4.PDOS.PlcToHw.digitalOutput_02 <-> Channel 2/Output
//     PlcTask Outputs/.P10_050_DO4.PDOS.PlcToHw.digitalOutput_03 <-> Channel 3/Output
//     PlcTask Outputs/.P10_050_DO4.PDOS.PlcToHw.digitalOutput_04 <-> Channel 4/Output
//     PlcTask Outputs/.P10_050_DO4.PDOS.PlcToHw.digitalOutput_05 <-> Channel 5/Output
//     PlcTask Outputs/.P10_050_DO4.PDOS.PlcToHw.digitalOutput_08 <-> Channel 8/Output
//     PlcTask Outputs/.P10_050_DO4.PDOS.PlcToHw.digitalOutput_09 <-> Channel 9/Output
//     PlcTask Outputs/.P10_050_DO4.PDOS.PlcToHw.digitalOutput_10 <-> Channel 10/Output
//     PlcTask Outputs/.P10_050_DO4.PDOS.PlcToHw.digitalOutput_11 <-> Channel 11/Output
//     PlcTask Outputs/.P10_050_DO4.PDOS.PlcToHw.digitalOutput_12 <-> Channel 12/Output
//     PlcTask Outputs/.P10_050_DO4.PDOS.PlcToHw.digitalOutput_13 <-> Channel 13/Output
//     PlcTask Outputs/.P10_050_DO4.PDOS.PlcToHw.digitalOutput_14 <-> Channel 14/Output
//     PlcTask Outputs/.P10_050_DO4.PDOS.PlcToHw.digitalOutput_15 <-> Channel 15/Output
//     PlcTask Outputs/.P10_050_DO4.PDOS.PlcToHw.digitalOutput_16 <-> Channel 16/Output
//     PlcTask Outputs/.P10_050_DO4.PDOS.PlcToHw.digitalOutput_06 <-> Channel 6/.P10_050_DO4.PDOS.PlcToHw.digitalOutput_06
//     PlcTask Outputs/.P10_050_DO4.PDOS.PlcToHw.digitalOutput_07 <-> Channel 7/.P10_050_DO4.PDOS.PlcToHw.digitalOutput_07
//   Plc_Prog/Plc_Prog Instance <-> ETH/+P10=050-BC2 - Press / Dryer PLC Cabinet/+P10=050-AI1 (EL3054)
//     PlcTask Inputs/.P10_050_AI1.PDOS.HwToPLC.Channel1/Status/Overrange <-> AI Standard Channel 1/Status/Overrange
//     PlcTask Inputs/.P10_050_AI1.PDOS.HwToPLC.Channel2/Status/Overrange <-> AI Standard Channel 2/Status/Overrange
//     PlcTask Inputs/.P10_050_AI1.PDOS.HwToPLC.Channel3/Status/Overrange <-> AI Standard Channel 3/Status/Overrange
//     PlcTask Inputs/.P10_050_AI1.PDOS.HwToPLC.Channel4/Status/Overrange <-> AI Standard Channel 4/Status/Overrange
//     PlcTask Inputs/.P10_050_AI1.PDOS.HwToPLC.Channel1/Status/Underrange <-> AI Standard Channel 1/Status/Underrange
//     PlcTask Inputs/.P10_050_AI1.PDOS.HwToPLC.Channel2/Status/Underrange <-> AI Standard Channel 2/Status/Underrange
//     PlcTask Inputs/.P10_050_AI1.PDOS.HwToPLC.Channel3/Status/Underrange <-> AI Standard Channel 3/Status/Underrange
//     PlcTask Inputs/.P10_050_AI1.PDOS.HwToPLC.Channel4/Status/Underrange <-> AI Standard Channel 4/Status/Underrange
//     PlcTask Inputs/.P10_050_AI1.PDOS.HwToPLC.Channel1/Value <-> AI Standard Channel 1/Value
//     PlcTask Inputs/.P10_050_AI1.PDOS.HwToPLC.Channel2/Value <-> AI Standard Channel 2/Value
//     PlcTask Inputs/.P10_050_AI1.PDOS.HwToPLC.Channel3/Value <-> AI Standard Channel 3/Value
//     PlcTask Inputs/.P10_050_AI1.PDOS.HwToPLC.Channel4/Value <-> AI Standard Channel 4/Value
//   Plc_Prog/Plc_Prog Instance <-> ETH/+P10=050-BC2 - Press / Dryer PLC Cabinet/+P10=050-AI2 (EL3204)
//     PlcTask Inputs/.P10_050_AI2.PDOS.HwToPLC.Channel1/Status/Overrange <-> RTD Inputs Channel 1/Status/Overrange
//     PlcTask Inputs/.P10_050_AI2.PDOS.HwToPLC.Channel2/Status/Overrange <-> RTD Inputs Channel 2/Status/Overrange
//     PlcTask Inputs/.P10_050_AI2.PDOS.HwToPLC.Channel3/Status/Overrange <-> RTD Inputs Channel 4/Status/Overrange
//     PlcTask Inputs/.P10_050_AI2.PDOS.HwToPLC.Channel4/Status/Overrange <-> RTD Inputs Channel 3/Status/Overrange
//     PlcTask Inputs/.P10_050_AI2.PDOS.HwToPLC.Channel1/Status/Underrange <-> RTD Inputs Channel 1/Status/Underrange
//     PlcTask Inputs/.P10_050_AI2.PDOS.HwToPLC.Channel2/Status/Underrange <-> RTD Inputs Channel 2/Status/Underrange
//     PlcTask Inputs/.P10_050_AI2.PDOS.HwToPLC.Channel3/Status/Underrange <-> RTD Inputs Channel 4/Status/Underrange
//     PlcTask Inputs/.P10_050_AI2.PDOS.HwToPLC.Channel4/Status/Underrange <-> RTD Inputs Channel 3/Status/Underrange
//     PlcTask Inputs/.P10_050_AI2.PDOS.HwToPLC.Channel1/Value <-> RTD Inputs Channel 1/Value
//     PlcTask Inputs/.P10_050_AI2.PDOS.HwToPLC.Channel2/Value <-> RTD Inputs Channel 2/Value
//     PlcTask Inputs/.P10_050_AI2.PDOS.HwToPLC.Channel3/Value <-> RTD Inputs Channel 3/Value
//     PlcTask Inputs/.P10_050_AI2.PDOS.HwToPLC.Channel4/Value <-> RTD Inputs Channel 4/Value
//   Plc_Prog/Plc_Prog Instance <-> ETH/+P10=050-BC2 - Press / Dryer PLC Cabinet/+P10=050-AO1(EL4024)
//     PlcTask Outputs/.P10_050_AO1.PDOS.HwToPLC.Channel1 <-> AO Outputs Channel 1/Analog output
//     PlcTask Outputs/.P10_050_AO1.PDOS.HwToPLC.Channel2 <-> AO Outputs Channel 2/Analog output
//     PlcTask Outputs/.P10_050_AO1.PDOS.HwToPLC.Channel3 <-> AO Outputs Channel 3/Analog output
//     PlcTask Outputs/.P10_050_AO1.PDOS.HwToPLC.Channel4 <-> AO Outputs Channel 4/Analog output
//   Plc_Prog/Plc_Prog Instance <-> ETH/+P11=400-UG1 - Second Press
//     PlcTask Inputs/.P11_400_UG01_SecondPress.PDOS.DrvToPLC.errorCode <-> 1st TxPDO Mapping/Error code
//     PlcTask Inputs/.P11_400_UG01_SecondPress.PDOS.DrvToPLC.modesOfOperationDisplay <-> 1st TxPDO Mapping/Mode Of Operation Display
//     PlcTask Inputs/.P11_400_UG01_SecondPress.PDOS.DrvToPLC.positionActualValue <-> 1st TxPDO Mapping/Position actual value
//     PlcTask Inputs/.P11_400_UG01_SecondPress.PDOS.DrvToPLC.statusWord <-> 1st TxPDO Mapping/Status Word
//     PlcTask Inputs/.P11_400_UG01_SecondPress.PDOS.DrvToPLC.torqueActualValue <-> 1st TxPDO Mapping/Torque actual value
//     PlcTask Inputs/.P11_400_UG01_SecondPress.PDOS.DrvToPLC.velocityActualValue <-> 1st TxPDO Mapping/Velocity actual value
//     PlcTask Outputs/.P11_400_UG01_SecondPress.PDOS.PlcToDrv.controlWord <-> 1st RxPDO Mapping/Control Word
//     PlcTask Outputs/.P11_400_UG01_SecondPress.PDOS.PlcToDrv.maxMotorSpeed <-> 1st RxPDO Mapping/Max motor speed
//     PlcTask Outputs/.P11_400_UG01_SecondPress.PDOS.PlcToDrv.maxTorque <-> 1st RxPDO Mapping/Target torque
//     PlcTask Outputs/.P11_400_UG01_SecondPress.PDOS.PlcToDrv.modesOfOperation <-> 1st RxPDO Mapping/Modes of operation
//     PlcTask Outputs/.P11_400_UG01_SecondPress.PDOS.PlcToDrv.vlTargetVelocity <-> 1st RxPDO Mapping/vl target velocity
//   Plc_Prog/Plc_Prog Instance <-> ETH/+P12=400-UG1 - First Press
//     PlcTask Inputs/.P12_400_UG01_FirstPress.PDOS.DrvToPLC.errorCode <-> 1st TxPDO Mapping/Error code
//     PlcTask Inputs/.P12_400_UG01_FirstPress.PDOS.DrvToPLC.modesOfOperationDisplay <-> 1st TxPDO Mapping/Mode Of Operation Display
//     PlcTask Inputs/.P12_400_UG01_FirstPress.PDOS.DrvToPLC.positionActualValue <-> 1st TxPDO Mapping/Position actual value
//     PlcTask Inputs/.P12_400_UG01_FirstPress.PDOS.DrvToPLC.statusWord <-> 1st TxPDO Mapping/Status Word
//     PlcTask Inputs/.P12_400_UG01_FirstPress.PDOS.DrvToPLC.torqueActualValue <-> 1st TxPDO Mapping/Torque actual value
//     PlcTask Inputs/.P12_400_UG01_FirstPress.PDOS.DrvToPLC.velocityActualValue <-> 1st TxPDO Mapping/Velocity actual value
//     PlcTask Outputs/.P12_400_UG01_FirstPress.PDOS.PlcToDrv.controlWord <-> 1st RxPDO Mapping/Control Word
//     PlcTask Outputs/.P12_400_UG01_FirstPress.PDOS.PlcToDrv.maxMotorSpeed <-> 1st RxPDO Mapping/Max motor speed
//     PlcTask Outputs/.P12_400_UG01_FirstPress.PDOS.PlcToDrv.maxTorque <-> 1st RxPDO Mapping/Target torque
//     PlcTask Outputs/.P12_400_UG01_FirstPress.PDOS.PlcToDrv.modesOfOperation <-> 1st RxPDO Mapping/Modes of operation
//     PlcTask Outputs/.P12_400_UG01_FirstPress.PDOS.PlcToDrv.vlTargetVelocity <-> 1st RxPDO Mapping/vl target velocity
//   Plc_Prog/Plc_Prog Instance <-> ETH/+P12=500-UG2 - Dryer Section GR1 - Lower GR1 Master
//     PlcTask Inputs/.P13_500_UG02_1GR_LowerMaster.PDOS.DrvToPLC.errorCode <-> 1st TxPDO Mapping/Error code
//     PlcTask Inputs/.P13_500_UG02_1GR_LowerMaster.PDOS.DrvToPLC.modesOfOperationDisplay <-> 1st TxPDO Mapping/Mode Of Operation Display
//     PlcTask Inputs/.P13_500_UG02_1GR_LowerMaster.PDOS.DrvToPLC.positionActualValue <-> 1st TxPDO Mapping/Position actual value
//     PlcTask Inputs/.P13_500_UG02_1GR_LowerMaster.PDOS.DrvToPLC.statusWord <-> 1st TxPDO Mapping/Status Word
//     PlcTask Inputs/.P13_500_UG02_1GR_LowerMaster.PDOS.DrvToPLC.torqueActualValue <-> 1st TxPDO Mapping/Torque actual value
//     PlcTask Inputs/.P13_500_UG02_1GR_LowerMaster.PDOS.DrvToPLC.velocityActualValue <-> 1st TxPDO Mapping/Velocity actual value
//     PlcTask Outputs/.P13_500_UG02_1GR_LowerMaster.PDOS.PlcToDrv.controlWord <-> 1st RxPDO Mapping/Control Word
//     PlcTask Outputs/.P13_500_UG02_1GR_LowerMaster.PDOS.PlcToDrv.maxMotorSpeed <-> 1st RxPDO Mapping/Max motor speed
//     PlcTask Outputs/.P13_500_UG02_1GR_LowerMaster.PDOS.PlcToDrv.maxTorque <-> 1st RxPDO Mapping/Target torque
//     PlcTask Outputs/.P13_500_UG02_1GR_LowerMaster.PDOS.PlcToDrv.modesOfOperation <-> 1st RxPDO Mapping/Modes of operation
//     PlcTask Outputs/.P13_500_UG02_1GR_LowerMaster.PDOS.PlcToDrv.vlTargetVelocity <-> 1st RxPDO Mapping/vl target velocity
//   Plc_Prog/Plc_Prog Instance <-> ETH/+P12=500-UG3 - Dryer Section GR1 - Upper Master
//     PlcTask Inputs/.P13_500_UG03_1GR_UpperMaster.PDOS.DrvToPLC.errorCode <-> 1st TxPDO Mapping/Error code
//     PlcTask Inputs/.P13_500_UG03_1GR_UpperMaster.PDOS.DrvToPLC.modesOfOperationDisplay <-> 1st TxPDO Mapping/Mode Of Operation Display
//     PlcTask Inputs/.P13_500_UG03_1GR_UpperMaster.PDOS.DrvToPLC.positionActualValue <-> 1st TxPDO Mapping/Position actual value
//     PlcTask Inputs/.P13_500_UG03_1GR_UpperMaster.PDOS.DrvToPLC.statusWord <-> 1st TxPDO Mapping/Status Word
//     PlcTask Inputs/.P13_500_UG03_1GR_UpperMaster.PDOS.DrvToPLC.torqueActualValue <-> 1st TxPDO Mapping/Torque actual value
//     PlcTask Inputs/.P13_500_UG03_1GR_UpperMaster.PDOS.DrvToPLC.velocityActualValue <-> 1st TxPDO Mapping/Velocity actual value
//     PlcTask Outputs/.P13_500_UG03_1GR_UpperMaster.PDOS.PlcToDrv.controlWord <-> 1st RxPDO Mapping/Control Word
//     PlcTask Outputs/.P13_500_UG03_1GR_UpperMaster.PDOS.PlcToDrv.maxMotorSpeed <-> 1st RxPDO Mapping/Max motor speed
//     PlcTask Outputs/.P13_500_UG03_1GR_UpperMaster.PDOS.PlcToDrv.maxTorque <-> 1st RxPDO Mapping/Target torque
//     PlcTask Outputs/.P13_500_UG03_1GR_UpperMaster.PDOS.PlcToDrv.modesOfOperation <-> 1st RxPDO Mapping/Modes of operation
//     PlcTask Outputs/.P13_500_UG03_1GR_UpperMaster.PDOS.PlcToDrv.vlTargetVelocity <-> 1st RxPDO Mapping/vl target velocity
//   Plc_Prog/Plc_Prog Instance <-> ETH/+P12=501-UG1 - Dryer Section  GR2 - Lower Slave
//     PlcTask Inputs/.P13_501_UG01_2GR_LowerSlave.PDOS.DrvToPLC.errorCode <-> 1st TxPDO Mapping/Error code
//     PlcTask Inputs/.P13_501_UG01_2GR_LowerSlave.PDOS.DrvToPLC.modesOfOperationDisplay <-> 1st TxPDO Mapping/Mode Of Operation Display
//     PlcTask Inputs/.P13_501_UG01_2GR_LowerSlave.PDOS.DrvToPLC.positionActualValue <-> 1st TxPDO Mapping/Position actual value
//     PlcTask Inputs/.P13_501_UG01_2GR_LowerSlave.PDOS.DrvToPLC.statusWord <-> 1st TxPDO Mapping/Status Word
//     PlcTask Inputs/.P13_501_UG01_2GR_LowerSlave.PDOS.DrvToPLC.torqueActualValue <-> 1st TxPDO Mapping/Torque actual value
//     PlcTask Inputs/.P13_501_UG01_2GR_LowerSlave.PDOS.DrvToPLC.velocityActualValue <-> 1st TxPDO Mapping/Velocity actual value
//     PlcTask Outputs/.P13_501_UG01_2GR_LowerSlave.PDOS.PlcToDrv.controlWord <-> 1st RxPDO Mapping/Control Word
//     PlcTask Outputs/.P13_501_UG01_2GR_LowerSlave.PDOS.PlcToDrv.maxMotorSpeed <-> 1st RxPDO Mapping/Max motor speed
//     PlcTask Outputs/.P13_501_UG01_2GR_LowerSlave.PDOS.PlcToDrv.maxTorque <-> 1st RxPDO Mapping/Target torque
//     PlcTask Outputs/.P13_501_UG01_2GR_LowerSlave.PDOS.PlcToDrv.modesOfOperation <-> 1st RxPDO Mapping/Modes of operation
//     PlcTask Outputs/.P13_501_UG01_2GR_LowerSlave.PDOS.PlcToDrv.vlTargetVelocity <-> 1st RxPDO Mapping/vl target velocity
//   Plc_Prog/Plc_Prog Instance <-> ETH/+P12=501-UG2 - Dryer Section GR2 - Upper Slave
//     PlcTask Inputs/.P13_501_UG02_2GR_UpperSlave.PDOS.DrvToPLC.errorCode <-> 1st TxPDO Mapping/Error code
//     PlcTask Inputs/.P13_501_UG02_2GR_UpperSlave.PDOS.DrvToPLC.modesOfOperationDisplay <-> 1st TxPDO Mapping/Mode Of Operation Display
//     PlcTask Inputs/.P13_501_UG02_2GR_UpperSlave.PDOS.DrvToPLC.positionActualValue <-> 1st TxPDO Mapping/Position actual value
//     PlcTask Inputs/.P13_501_UG02_2GR_UpperSlave.PDOS.DrvToPLC.statusWord <-> 1st TxPDO Mapping/Status Word
//     PlcTask Inputs/.P13_501_UG02_2GR_UpperSlave.PDOS.DrvToPLC.torqueActualValue <-> 1st TxPDO Mapping/Torque actual value
//     PlcTask Inputs/.P13_501_UG02_2GR_UpperSlave.PDOS.DrvToPLC.velocityActualValue <-> 1st TxPDO Mapping/Velocity actual value
//     PlcTask Outputs/.P13_501_UG02_2GR_UpperSlave.PDOS.PlcToDrv.controlWord <-> 1st RxPDO Mapping/Control Word
//     PlcTask Outputs/.P13_501_UG02_2GR_UpperSlave.PDOS.PlcToDrv.maxMotorSpeed <-> 1st RxPDO Mapping/Max motor speed
//     PlcTask Outputs/.P13_501_UG02_2GR_UpperSlave.PDOS.PlcToDrv.maxTorque <-> 1st RxPDO Mapping/Target torque
//     PlcTask Outputs/.P13_501_UG02_2GR_UpperSlave.PDOS.PlcToDrv.modesOfOperation <-> 1st RxPDO Mapping/Modes of operation
//     PlcTask Outputs/.P13_501_UG02_2GR_UpperSlave.PDOS.PlcToDrv.vlTargetVelocity <-> 1st RxPDO Mapping/vl target velocity
//   Plc_Prog/Plc_Prog Instance <-> ETH/+P12=501-UG3 - Dryer Section GR2 - Lower Master
//     PlcTask Inputs/.P13_501_UG03_2GR_LowerMaster.PDOS.DrvToPLC.errorCode <-> 1st TxPDO Mapping/Error code
//     PlcTask Inputs/.P13_501_UG03_2GR_LowerMaster.PDOS.DrvToPLC.modesOfOperationDisplay <-> 1st TxPDO Mapping/Mode Of Operation Display
//     PlcTask Inputs/.P13_501_UG03_2GR_LowerMaster.PDOS.DrvToPLC.positionActualValue <-> 1st TxPDO Mapping/Position actual value
//     PlcTask Inputs/.P13_501_UG03_2GR_LowerMaster.PDOS.DrvToPLC.statusWord <-> 1st TxPDO Mapping/Status Word
//     PlcTask Inputs/.P13_501_UG03_2GR_LowerMaster.PDOS.DrvToPLC.torqueActualValue <-> 1st TxPDO Mapping/Torque actual value
//     PlcTask Inputs/.P13_501_UG03_2GR_LowerMaster.PDOS.DrvToPLC.velocityActualValue <-> 1st TxPDO Mapping/Velocity actual value
//     PlcTask Outputs/.P13_501_UG03_2GR_LowerMaster.PDOS.PlcToDrv.controlWord <-> 1st RxPDO Mapping/Control Word
//     PlcTask Outputs/.P13_501_UG03_2GR_LowerMaster.PDOS.PlcToDrv.maxMotorSpeed <-> 1st RxPDO Mapping/Max motor speed
//     PlcTask Outputs/.P13_501_UG03_2GR_LowerMaster.PDOS.PlcToDrv.maxTorque <-> 1st RxPDO Mapping/Target torque
//     PlcTask Outputs/.P13_501_UG03_2GR_LowerMaster.PDOS.PlcToDrv.modesOfOperation <-> 1st RxPDO Mapping/Modes of operation
//     PlcTask Outputs/.P13_501_UG03_2GR_LowerMaster.PDOS.PlcToDrv.vlTargetVelocity <-> 1st RxPDO Mapping/vl target velocity
//   Plc_Prog/Plc_Prog Instance <-> ETH/+P13=500-UG1 - Dryer Section GR1 - Upper GR1 Slave
//     PlcTask Inputs/.P13_500_UG01_1GR_UpperSlave.PDOS.DrvToPLC.errorCode <-> 1st TxPDO Mapping/Error code
//     PlcTask Inputs/.P13_500_UG01_1GR_UpperSlave.PDOS.DrvToPLC.modesOfOperationDisplay <-> 1st TxPDO Mapping/Mode Of Operation Display
//     PlcTask Inputs/.P13_500_UG01_1GR_UpperSlave.PDOS.DrvToPLC.positionActualValue <-> 1st TxPDO Mapping/Position actual value
//     PlcTask Inputs/.P13_500_UG01_1GR_UpperSlave.PDOS.DrvToPLC.statusWord <-> 1st TxPDO Mapping/Status Word
//     PlcTask Inputs/.P13_500_UG01_1GR_UpperSlave.PDOS.DrvToPLC.torqueActualValue <-> 1st TxPDO Mapping/Torque actual value
//     PlcTask Inputs/.P13_500_UG01_1GR_UpperSlave.PDOS.DrvToPLC.velocityActualValue <-> 1st TxPDO Mapping/Velocity actual value
//     PlcTask Outputs/.P13_500_UG01_1GR_UpperSlave.PDOS.PlcToDrv.controlWord <-> 1st RxPDO Mapping/Control Word
//     PlcTask Outputs/.P13_500_UG01_1GR_UpperSlave.PDOS.PlcToDrv.maxMotorSpeed <-> 1st RxPDO Mapping/Max motor speed
//     PlcTask Outputs/.P13_500_UG01_1GR_UpperSlave.PDOS.PlcToDrv.maxTorque <-> 1st RxPDO Mapping/Target torque
//     PlcTask Outputs/.P13_500_UG01_1GR_UpperSlave.PDOS.PlcToDrv.modesOfOperation <-> 1st RxPDO Mapping/Modes of operation
//     PlcTask Outputs/.P13_500_UG01_1GR_UpperSlave.PDOS.PlcToDrv.vlTargetVelocity <-> 1st RxPDO Mapping/vl target velocity
//   Plc_Prog/Plc_Prog Instance <-> ETH/+P13=501-UG1 - Dryer Section GR2 - Upper Master
//     PlcTask Inputs/.P14_501_UG01_2GR_UpperMaster.PDOS.DrvToPLC.errorCode <-> 1st TxPDO Mapping/Error code
//     PlcTask Inputs/.P14_501_UG01_2GR_UpperMaster.PDOS.DrvToPLC.modesOfOperationDisplay <-> 1st TxPDO Mapping/Mode Of Operation Display
//     PlcTask Inputs/.P14_501_UG01_2GR_UpperMaster.PDOS.DrvToPLC.positionActualValue <-> 1st TxPDO Mapping/Position actual value
//     PlcTask Inputs/.P14_501_UG01_2GR_UpperMaster.PDOS.DrvToPLC.statusWord <-> 1st TxPDO Mapping/Status Word
//     PlcTask Inputs/.P14_501_UG01_2GR_UpperMaster.PDOS.DrvToPLC.torqueActualValue <-> 1st TxPDO Mapping/Torque actual value
//     PlcTask Inputs/.P14_501_UG01_2GR_UpperMaster.PDOS.DrvToPLC.velocityActualValue <-> 1st TxPDO Mapping/Velocity actual value
//     PlcTask Outputs/.P14_501_UG01_2GR_UpperMaster.PDOS.PlcToDrv.controlWord <-> 1st RxPDO Mapping/Control Word
//     PlcTask Outputs/.P14_501_UG01_2GR_UpperMaster.PDOS.PlcToDrv.maxMotorSpeed <-> 1st RxPDO Mapping/Max motor speed
//     PlcTask Outputs/.P14_501_UG01_2GR_UpperMaster.PDOS.PlcToDrv.maxTorque <-> 1st RxPDO Mapping/Target torque
//     PlcTask Outputs/.P14_501_UG01_2GR_UpperMaster.PDOS.PlcToDrv.modesOfOperation <-> 1st RxPDO Mapping/Modes of operation
//     PlcTask Outputs/.P14_501_UG01_2GR_UpperMaster.PDOS.PlcToDrv.vlTargetVelocity <-> 1st RxPDO Mapping/vl target velocity
//   Plc_Prog/Plc_Prog Instance <-> ETH/+P13=502-UG2 - Dryer Section GR3 - Lower Slave
//     PlcTask Inputs/.P14_502_UG01_3GR_LowerSlave.PDOS.DrvToPLC.errorCode <-> 1st TxPDO Mapping/Error code
//     PlcTask Inputs/.P14_502_UG01_3GR_LowerSlave.PDOS.DrvToPLC.modesOfOperationDisplay <-> 1st TxPDO Mapping/Mode Of Operation Display
//     PlcTask Inputs/.P14_502_UG01_3GR_LowerSlave.PDOS.DrvToPLC.positionActualValue <-> 1st TxPDO Mapping/Position actual value
//     PlcTask Inputs/.P14_502_UG01_3GR_LowerSlave.PDOS.DrvToPLC.statusWord <-> 1st TxPDO Mapping/Status Word
//     PlcTask Inputs/.P14_502_UG01_3GR_LowerSlave.PDOS.DrvToPLC.torqueActualValue <-> 1st TxPDO Mapping/Torque actual value
//     PlcTask Inputs/.P14_502_UG01_3GR_LowerSlave.PDOS.DrvToPLC.velocityActualValue <-> 1st TxPDO Mapping/Velocity actual value
//     PlcTask Outputs/.P14_502_UG01_3GR_LowerSlave.PDOS.PlcToDrv.controlWord <-> 1st RxPDO Mapping/Control Word
//     PlcTask Outputs/.P14_502_UG01_3GR_LowerSlave.PDOS.PlcToDrv.maxMotorSpeed <-> 1st RxPDO Mapping/Max motor speed
//     PlcTask Outputs/.P14_502_UG01_3GR_LowerSlave.PDOS.PlcToDrv.maxTorque <-> 1st RxPDO Mapping/Target torque
//     PlcTask Outputs/.P14_502_UG01_3GR_LowerSlave.PDOS.PlcToDrv.modesOfOperation <-> 1st RxPDO Mapping/Modes of operation
//     PlcTask Outputs/.P14_502_UG01_3GR_LowerSlave.PDOS.PlcToDrv.vlTargetVelocity <-> 1st RxPDO Mapping/vl target velocity
//   Plc_Prog/Plc_Prog Instance <-> ETH/+P13=502-UG2 - Dryer Section GR3 - Upper Slave
//     PlcTask Inputs/.P14_502_UG02_3GR_UpperSlave.PDOS.DrvToPLC.errorCode <-> 1st TxPDO Mapping/Error code
//     PlcTask Inputs/.P14_502_UG02_3GR_UpperSlave.PDOS.DrvToPLC.modesOfOperationDisplay <-> 1st TxPDO Mapping/Mode Of Operation Display
//     PlcTask Inputs/.P14_502_UG02_3GR_UpperSlave.PDOS.DrvToPLC.positionActualValue <-> 1st TxPDO Mapping/Position actual value
//     PlcTask Inputs/.P14_502_UG02_3GR_UpperSlave.PDOS.DrvToPLC.statusWord <-> 1st TxPDO Mapping/Status Word
//     PlcTask Inputs/.P14_502_UG02_3GR_UpperSlave.PDOS.DrvToPLC.torqueActualValue <-> 1st TxPDO Mapping/Torque actual value
//     PlcTask Inputs/.P14_502_UG02_3GR_UpperSlave.PDOS.DrvToPLC.velocityActualValue <-> 1st TxPDO Mapping/Velocity actual value
//     PlcTask Outputs/.P14_502_UG02_3GR_UpperSlave.PDOS.PlcToDrv.controlWord <-> 1st RxPDO Mapping/Control Word
//     PlcTask Outputs/.P14_502_UG02_3GR_UpperSlave.PDOS.PlcToDrv.maxMotorSpeed <-> 1st RxPDO Mapping/Max motor speed
//     PlcTask Outputs/.P14_502_UG02_3GR_UpperSlave.PDOS.PlcToDrv.maxTorque <-> 1st RxPDO Mapping/Target torque
//     PlcTask Outputs/.P14_502_UG02_3GR_UpperSlave.PDOS.PlcToDrv.modesOfOperation <-> 1st RxPDO Mapping/Modes of operation
//     PlcTask Outputs/.P14_502_UG02_3GR_UpperSlave.PDOS.PlcToDrv.vlTargetVelocity <-> 1st RxPDO Mapping/vl target velocity
//   Plc_Prog/Plc_Prog Instance <-> ETH/+P13=502-UG3 - Dryer Section GR3 - Lower Master
//     PlcTask Inputs/.P14_502_UG03_3GR_LowerMaster.PDOS.DrvToPLC.errorCode <-> 1st TxPDO Mapping/Error code
//     PlcTask Inputs/.P14_502_UG03_3GR_LowerMaster.PDOS.DrvToPLC.modesOfOperationDisplay <-> 1st TxPDO Mapping/Mode Of Operation Display
//     PlcTask Inputs/.P14_502_UG03_3GR_LowerMaster.PDOS.DrvToPLC.positionActualValue <-> 1st TxPDO Mapping/Position actual value
//     PlcTask Inputs/.P14_502_UG03_3GR_LowerMaster.PDOS.DrvToPLC.statusWord <-> 1st TxPDO Mapping/Status Word
//     PlcTask Inputs/.P14_502_UG03_3GR_LowerMaster.PDOS.DrvToPLC.torqueActualValue <-> 1st TxPDO Mapping/Torque actual value
//     PlcTask Inputs/.P14_502_UG03_3GR_LowerMaster.PDOS.DrvToPLC.velocityActualValue <-> 1st TxPDO Mapping/Velocity actual value
//     PlcTask Outputs/.P14_502_UG03_3GR_LowerMaster.PDOS.PlcToDrv.controlWord <-> 1st RxPDO Mapping/Control Word
//     PlcTask Outputs/.P14_502_UG03_3GR_LowerMaster.PDOS.PlcToDrv.maxMotorSpeed <-> 1st RxPDO Mapping/Max motor speed
//     PlcTask Outputs/.P14_502_UG03_3GR_LowerMaster.PDOS.PlcToDrv.maxTorque <-> 1st RxPDO Mapping/Target torque
//     PlcTask Outputs/.P14_502_UG03_3GR_LowerMaster.PDOS.PlcToDrv.modesOfOperation <-> 1st RxPDO Mapping/Modes of operation
//     PlcTask Outputs/.P14_502_UG03_3GR_LowerMaster.PDOS.PlcToDrv.vlTargetVelocity <-> 1st RxPDO Mapping/vl target velocity
//   Plc_Prog/Plc_Prog Instance <-> ETH/+P13=502-UG4 - Dryer Section GR3 - Upper Master
//     PlcTask Inputs/.P14_502_UG04_3GR_UpperMaster.PDOS.DrvToPLC.errorCode <-> 1st TxPDO Mapping/Error code
//     PlcTask Inputs/.P14_502_UG04_3GR_UpperMaster.PDOS.DrvToPLC.modesOfOperationDisplay <-> 1st TxPDO Mapping/Mode Of Operation Display
//     PlcTask Inputs/.P14_502_UG04_3GR_UpperMaster.PDOS.DrvToPLC.positionActualValue <-> 1st TxPDO Mapping/Position actual value
//     PlcTask Inputs/.P14_502_UG04_3GR_UpperMaster.PDOS.DrvToPLC.statusWord <-> 1st TxPDO Mapping/Status Word
//     PlcTask Inputs/.P14_502_UG04_3GR_UpperMaster.PDOS.DrvToPLC.torqueActualValue <-> 1st TxPDO Mapping/Torque actual value
//     PlcTask Inputs/.P14_502_UG04_3GR_UpperMaster.PDOS.DrvToPLC.velocityActualValue <-> 1st TxPDO Mapping/Velocity actual value
//     PlcTask Outputs/.P14_502_UG04_3GR_UpperMaster.PDOS.PlcToDrv.controlWord <-> 1st RxPDO Mapping/Control Word
//     PlcTask Outputs/.P14_502_UG04_3GR_UpperMaster.PDOS.PlcToDrv.maxMotorSpeed <-> 1st RxPDO Mapping/Max motor speed
//     PlcTask Outputs/.P14_502_UG04_3GR_UpperMaster.PDOS.PlcToDrv.maxTorque <-> 1st RxPDO Mapping/Target torque
//     PlcTask Outputs/.P14_502_UG04_3GR_UpperMaster.PDOS.PlcToDrv.modesOfOperation <-> 1st RxPDO Mapping/Modes of operation
//     PlcTask Outputs/.P14_502_UG04_3GR_UpperMaster.PDOS.PlcToDrv.vlTargetVelocity <-> 1st RxPDO Mapping/vl target velocity
//   Plc_Prog/Plc_Prog Instance <-> ETH/+P14=600-UG1 - Winder
//     PlcTask Inputs/.P15_600_UG01_Rewinder.PDOS.DrvToPLC.errorCode <-> 1st TxPDO Mapping/Error code
//     PlcTask Inputs/.P15_600_UG01_Rewinder.PDOS.DrvToPLC.modesOfOperationDisplay <-> 1st TxPDO Mapping/Mode Of Operation Display
//     PlcTask Inputs/.P15_600_UG01_Rewinder.PDOS.DrvToPLC.positionActualValue <-> 1st TxPDO Mapping/Position actual value
//     PlcTask Inputs/.P15_600_UG01_Rewinder.PDOS.DrvToPLC.statusWord <-> 1st TxPDO Mapping/Status Word
//     PlcTask Inputs/.P15_600_UG01_Rewinder.PDOS.DrvToPLC.torqueActualValue <-> 1st TxPDO Mapping/Torque actual value
//     PlcTask Inputs/.P15_600_UG01_Rewinder.PDOS.DrvToPLC.velocityActualValue <-> 1st TxPDO Mapping/Velocity actual value
//     PlcTask Outputs/.P15_600_UG01_Rewinder.PDOS.PlcToDrv.controlWord <-> 1st RxPDO Mapping/Control Word
//     PlcTask Outputs/.P15_600_UG01_Rewinder.PDOS.PlcToDrv.maxMotorSpeed <-> 1st RxPDO Mapping/Max motor speed
//     PlcTask Outputs/.P15_600_UG01_Rewinder.PDOS.PlcToDrv.maxTorque <-> 1st RxPDO Mapping/Target torque
//     PlcTask Outputs/.P15_600_UG01_Rewinder.PDOS.PlcToDrv.modesOfOperation <-> 1st RxPDO Mapping/Modes of operation
//     PlcTask Outputs/.P15_600_UG01_Rewinder.PDOS.PlcToDrv.vlTargetVelocity <-> 1st RxPDO Mapping/vl target velocity
//   Plc_Prog/Plc_Prog Instance <-> ETH/+P2=100-UG1 - Drive Roll
//     PlcTask Inputs/.P1_300_UG06_TractionRoll.PDOS.DrvToPLC.errorCode <-> 1st TxPDO Mapping/Error code
//     PlcTask Inputs/.P1_300_UG06_TractionRoll.PDOS.DrvToPLC.modesOfOperationDisplay <-> 1st TxPDO Mapping/Mode Of Operation Display
//     PlcTask Inputs/.P1_300_UG06_TractionRoll.PDOS.DrvToPLC.positionActualValue <-> 1st TxPDO Mapping/Position actual value
//     PlcTask Inputs/.P1_300_UG06_TractionRoll.PDOS.DrvToPLC.statusWord <-> 1st TxPDO Mapping/Status Word
//     PlcTask Inputs/.P1_300_UG06_TractionRoll.PDOS.DrvToPLC.torqueActualValue <-> 1st TxPDO Mapping/Torque actual value
//     PlcTask Inputs/.P1_300_UG06_TractionRoll.PDOS.DrvToPLC.velocityActualValue <-> 1st TxPDO Mapping/Velocity actual value
//     PlcTask Outputs/.P1_300_UG06_TractionRoll.PDOS.PlcToDrv.controlWord <-> 1st RxPDO Mapping/Control Word
//     PlcTask Outputs/.P1_300_UG06_TractionRoll.PDOS.PlcToDrv.maxMotorSpeed <-> 1st RxPDO Mapping/Max motor speed
//     PlcTask Outputs/.P1_300_UG06_TractionRoll.PDOS.PlcToDrv.maxTorque <-> 1st RxPDO Mapping/Max torque
//     PlcTask Outputs/.P1_300_UG06_TractionRoll.PDOS.PlcToDrv.modesOfOperation <-> 1st RxPDO Mapping/Modes of operation
//     PlcTask Outputs/.P1_300_UG06_TractionRoll.PDOS.PlcToDrv.vlTargetVelocity <-> 1st RxPDO Mapping/vl target velocity
//   Plc_Prog/Plc_Prog Instance <-> ETH/+P3=100-UG1 - CouchPit
//     PlcTask Inputs/.P1_100_UG04.PDOS.DrvToPLC.errorCode <-> 1st TxPDO Mapping/Error code
//     PlcTask Inputs/.P1_100_UG04.PDOS.DrvToPLC.modesOfOperationDisplay <-> 1st TxPDO Mapping/Mode Of Operation Display
//     PlcTask Inputs/.P1_100_UG04.PDOS.DrvToPLC.positionActualValue <-> 1st TxPDO Mapping/Position actual value
//     PlcTask Inputs/.P1_100_UG04.PDOS.DrvToPLC.statusWord <-> 1st TxPDO Mapping/Status Word
//     PlcTask Inputs/.P1_100_UG04.PDOS.DrvToPLC.torqueActualValue <-> 1st TxPDO Mapping/Torque actual value
//     PlcTask Inputs/.P1_100_UG04.PDOS.DrvToPLC.velocityActualValue <-> 1st TxPDO Mapping/Velocity actual value
//     PlcTask Outputs/.P1_100_UG04.PDOS.PlcToDrv.controlWord <-> 1st RxPDO Mapping/Control Word
//     PlcTask Outputs/.P1_100_UG04.PDOS.PlcToDrv.maxMotorSpeed <-> 1st RxPDO Mapping/Max motor speed
//     PlcTask Outputs/.P1_100_UG04.PDOS.PlcToDrv.maxTorque <-> 1st RxPDO Mapping/Max torque
//     PlcTask Outputs/.P1_100_UG04.PDOS.PlcToDrv.modesOfOperation <-> 1st RxPDO Mapping/Modes of operation
//     PlcTask Outputs/.P1_100_UG04.PDOS.PlcToDrv.vlTargetVelocity <-> 1st RxPDO Mapping/vl target velocity
//   Plc_Prog/Plc_Prog Instance <-> ETH/+P3=100-UG1 - SuctionRoll
//     PlcTask Inputs/.P1_100_UG03_SuctionRoll.PDOS.DrvToPLC.errorCode <-> 1st TxPDO Mapping/Error code
//     PlcTask Inputs/.P1_100_UG03_SuctionRoll.PDOS.DrvToPLC.modesOfOperationDisplay <-> 1st TxPDO Mapping/Mode Of Operation Display
//     PlcTask Inputs/.P1_100_UG03_SuctionRoll.PDOS.DrvToPLC.positionActualValue <-> 1st TxPDO Mapping/Position actual value
//     PlcTask Inputs/.P1_100_UG03_SuctionRoll.PDOS.DrvToPLC.statusWord <-> 1st TxPDO Mapping/Status Word
//     PlcTask Inputs/.P1_100_UG03_SuctionRoll.PDOS.DrvToPLC.torqueActualValue <-> 1st TxPDO Mapping/Torque actual value
//     PlcTask Inputs/.P1_100_UG03_SuctionRoll.PDOS.DrvToPLC.velocityActualValue <-> 1st TxPDO Mapping/Velocity actual value
//     PlcTask Outputs/.P1_100_UG03_SuctionRoll.PDOS.PlcToDrv.controlWord <-> 1st RxPDO Mapping/Control Word
//     PlcTask Outputs/.P1_100_UG03_SuctionRoll.PDOS.PlcToDrv.maxMotorSpeed <-> 1st RxPDO Mapping/Max motor speed
//     PlcTask Outputs/.P1_100_UG03_SuctionRoll.PDOS.PlcToDrv.maxTorque <-> 1st RxPDO Mapping/Target torque
//     PlcTask Outputs/.P1_100_UG03_SuctionRoll.PDOS.PlcToDrv.modesOfOperation <-> 1st RxPDO Mapping/Modes of operation
//     PlcTask Outputs/.P1_100_UG03_SuctionRoll.PDOS.PlcToDrv.vlTargetVelocity <-> 1st RxPDO Mapping/vl target velocity
//   Plc_Prog/Plc_Prog Instance <-> ETH/+P3=100-UG2 - Stock pump
//     PlcTask Inputs/.P1_100_UG05.PDOS.DrvToPLC.errorCode <-> 1st TxPDO Mapping/Error code
//     PlcTask Inputs/.P1_100_UG05.PDOS.DrvToPLC.modesOfOperationDisplay <-> 1st TxPDO Mapping/Mode Of Operation Display
//     PlcTask Inputs/.P1_100_UG05.PDOS.DrvToPLC.positionActualValue <-> 1st TxPDO Mapping/Position actual value
//     PlcTask Inputs/.P1_100_UG05.PDOS.DrvToPLC.statusWord <-> 1st TxPDO Mapping/Status Word
//     PlcTask Inputs/.P1_100_UG05.PDOS.DrvToPLC.torqueActualValue <-> 1st TxPDO Mapping/Torque actual value
//     PlcTask Inputs/.P1_100_UG05.PDOS.DrvToPLC.velocityActualValue <-> 1st TxPDO Mapping/Velocity actual value
//     PlcTask Outputs/.P1_100_UG05.PDOS.PlcToDrv.controlWord <-> 1st RxPDO Mapping/Control Word
//     PlcTask Outputs/.P1_100_UG05.PDOS.PlcToDrv.maxMotorSpeed <-> 1st RxPDO Mapping/Max motor speed
//     PlcTask Outputs/.P1_100_UG05.PDOS.PlcToDrv.maxTorque <-> 1st RxPDO Mapping/Max torque
//     PlcTask Outputs/.P1_100_UG05.PDOS.PlcToDrv.modesOfOperation <-> 1st RxPDO Mapping/Modes of operation
//     PlcTask Outputs/.P1_100_UG05.PDOS.PlcToDrv.vlTargetVelocity <-> 1st RxPDO Mapping/vl target velocity
//   Plc_Prog/Plc_Prog Instance <-> ETH/+P3=300-UG1 - WirePit Pump
//     PlcTask Inputs/.P1_100_UG02.PDOS.DrvToPLC.errorCode <-> 1st TxPDO Mapping/Error code
//     PlcTask Inputs/.P1_100_UG02.PDOS.DrvToPLC.modesOfOperationDisplay <-> 1st TxPDO Mapping/Mode Of Operation Display
//     PlcTask Inputs/.P1_100_UG02.PDOS.DrvToPLC.positionActualValue <-> 1st TxPDO Mapping/Position actual value
//     PlcTask Inputs/.P1_100_UG02.PDOS.DrvToPLC.statusWord <-> 1st TxPDO Mapping/Status Word
//     PlcTask Inputs/.P1_100_UG02.PDOS.DrvToPLC.torqueActualValue <-> 1st TxPDO Mapping/Torque actual value
//     PlcTask Inputs/.P1_100_UG02.PDOS.DrvToPLC.velocityActualValue <-> 1st TxPDO Mapping/Velocity actual value
//     PlcTask Outputs/.P1_100_UG02.PDOS.PlcToDrv.controlWord <-> 1st RxPDO Mapping/Control Word
//     PlcTask Outputs/.P1_100_UG02.PDOS.PlcToDrv.maxMotorSpeed <-> 1st RxPDO Mapping/Max motor speed
//     PlcTask Outputs/.P1_100_UG02.PDOS.PlcToDrv.maxTorque <-> 1st RxPDO Mapping/Max torque
//     PlcTask Outputs/.P1_100_UG02.PDOS.PlcToDrv.modesOfOperation <-> 1st RxPDO Mapping/Modes of operation
//     PlcTask Outputs/.P1_100_UG02.PDOS.PlcToDrv.vlTargetVelocity <-> 1st RxPDO Mapping/vl target velocity
//   Plc_Prog/Plc_Prog Instance <-> ETH/+P4=300-UG1 - Mix Pump
//     PlcTask Inputs/.P1_100_UG01.PDOS.DrvToPLC.errorCode <-> 1st TxPDO Mapping/Error code
//     PlcTask Inputs/.P1_100_UG01.PDOS.DrvToPLC.modesOfOperationDisplay <-> 1st TxPDO Mapping/Mode Of Operation Display
//     PlcTask Inputs/.P1_100_UG01.PDOS.DrvToPLC.positionActualValue <-> 1st TxPDO Mapping/Position actual value
//     PlcTask Inputs/.P1_100_UG01.PDOS.DrvToPLC.statusWord <-> 1st TxPDO Mapping/Status Word
//     PlcTask Inputs/.P1_100_UG01.PDOS.DrvToPLC.torqueActualValue <-> 1st TxPDO Mapping/Torque actual value
//     PlcTask Inputs/.P1_100_UG01.PDOS.DrvToPLC.velocityActualValue <-> 1st TxPDO Mapping/Velocity actual value
//     PlcTask Outputs/.P1_100_UG01.PDOS.PlcToDrv.controlWord <-> 1st RxPDO Mapping/Control Word
//     PlcTask Outputs/.P1_100_UG01.PDOS.PlcToDrv.maxMotorSpeed <-> 1st RxPDO Mapping/Max motor speed
//     PlcTask Outputs/.P1_100_UG01.PDOS.PlcToDrv.maxTorque <-> 1st RxPDO Mapping/Max torque
//     PlcTask Outputs/.P1_100_UG01.PDOS.PlcToDrv.modesOfOperation <-> 1st RxPDO Mapping/Modes of operation
//     PlcTask Outputs/.P1_100_UG01.PDOS.PlcToDrv.vlTargetVelocity <-> 1st RxPDO Mapping/vl target velocity
//   Plc_Prog/Plc_Prog Instance <-> ETH/+P5=050-BC1 - PLC Cabinet/+P5=050-DI1 (EL1809)
//     PlcTask Inputs/.P1_050_DI1.PDOS.digitalInput_01 <-> Channel 1/Input
//     PlcTask Inputs/.P1_050_DI1.PDOS.digitalInput_02 <-> Channel 2/Input
//     PlcTask Inputs/.P1_050_DI1.PDOS.digitalInput_03 <-> Channel 3/Input
//     PlcTask Inputs/.P1_050_DI1.PDOS.digitalInput_04 <-> Channel 4/Input
//     PlcTask Inputs/.P1_050_DI1.PDOS.digitalInput_05 <-> Channel 5/Input
//     PlcTask Inputs/.P1_050_DI1.PDOS.digitalInput_06 <-> Channel 6/Input
//     PlcTask Inputs/.P1_050_DI1.PDOS.digitalInput_07 <-> Channel 7/Input
//     PlcTask Inputs/.P1_050_DI1.PDOS.digitalInput_08 <-> Channel 8/Input
//     PlcTask Inputs/.P1_050_DI1.PDOS.digitalInput_09 <-> Channel 9/Input
//     PlcTask Inputs/.P1_050_DI1.PDOS.digitalInput_10 <-> Channel 10/Input
//     PlcTask Inputs/.P1_050_DI1.PDOS.digitalInput_11 <-> Channel 11/Input
//     PlcTask Inputs/.P1_050_DI1.PDOS.digitalInput_12 <-> Channel 12/Input
//     PlcTask Inputs/.P1_050_DI1.PDOS.digitalInput_13 <-> Channel 13/Input
//     PlcTask Inputs/.P1_050_DI1.PDOS.digitalInput_14 <-> Channel 14/Input
//     PlcTask Inputs/.P1_050_DI1.PDOS.digitalInput_15 <-> Channel 15/Input
//     PlcTask Inputs/.P1_050_DI1.PDOS.digitalInput_16 <-> Channel 16/Input
//   Plc_Prog/Plc_Prog Instance <-> ETH/+P5=050-BC1 - PLC Cabinet/+P5=050-DI2 (EL1809)
//     PlcTask Inputs/.P1_050_DI2.PDOS.digitalInput_01 <-> Channel 1/Input
//     PlcTask Inputs/.P1_050_DI2.PDOS.digitalInput_02 <-> Channel 2/Input
//     PlcTask Inputs/.P1_050_DI2.PDOS.digitalInput_03 <-> Channel 3/Input
//     PlcTask Inputs/.P1_050_DI2.PDOS.digitalInput_04 <-> Channel 4/Input
//     PlcTask Inputs/.P1_050_DI2.PDOS.digitalInput_05 <-> Channel 5/Input
//     PlcTask Inputs/.P1_050_DI2.PDOS.digitalInput_06 <-> Channel 6/Input
//     PlcTask Inputs/.P1_050_DI2.PDOS.digitalInput_07 <-> Channel 7/Input
//     PlcTask Inputs/.P1_050_DI2.PDOS.digitalInput_08 <-> Channel 8/Input
//     PlcTask Inputs/.P1_050_DI2.PDOS.digitalInput_09 <-> Channel 9/Input
//     PlcTask Inputs/.P1_050_DI2.PDOS.digitalInput_10 <-> Channel 10/Input
//     PlcTask Inputs/.P1_050_DI2.PDOS.digitalInput_13 <-> Channel 13/Input
//     PlcTask Inputs/.P1_050_DI2.PDOS.digitalInput_14 <-> Channel 14/Input
//     PlcTask Inputs/.P1_050_DI2.PDOS.digitalInput_15 <-> Channel 15/Input
//     PlcTask Inputs/.P1_050_DI2.PDOS.digitalInput_16 <-> Channel 16/Input
//     PlcTask Inputs/.P1_050_DI2.PDOS.digitalInput_11 <-> Channel 11/.P1_050_DI2.PDOS.digitalInput_11
//     PlcTask Inputs/.P1_050_DI2.PDOS.digitalInput_12 <-> Channel 12/.P1_050_DI2.PDOS.digitalInput_12
//   Plc_Prog/Plc_Prog Instance <-> ETH/+P5=050-BC1 - PLC Cabinet/+P5=050-DI3 (EL1809)
//     PlcTask Inputs/.P1_050_DI3.PDOS.digitalInput_01 <-> Channel 1/Input
//     PlcTask Inputs/.P1_050_DI3.PDOS.digitalInput_02 <-> Channel 2/Input
//     PlcTask Inputs/.P1_050_DI3.PDOS.digitalInput_03 <-> Channel 3/Input
//     PlcTask Inputs/.P1_050_DI3.PDOS.digitalInput_04 <-> Channel 4/Input
//     PlcTask Inputs/.P1_050_DI3.PDOS.digitalInput_05 <-> Channel 5/Input
//     PlcTask Inputs/.P1_050_DI3.PDOS.digitalInput_06 <-> Channel 6/Input
//     PlcTask Inputs/.P1_050_DI3.PDOS.digitalInput_07 <-> Channel 7/Input
//     PlcTask Inputs/.P1_050_DI3.PDOS.digitalInput_08 <-> Channel 8/Input
//     PlcTask Inputs/.P1_050_DI3.PDOS.digitalInput_09 <-> Channel 9/Input
//     PlcTask Inputs/.P1_050_DI3.PDOS.digitalInput_10 <-> Channel 10/Input
//     PlcTask Inputs/.P1_050_DI3.PDOS.digitalInput_11 <-> Channel 11/Input
//     PlcTask Inputs/.P1_050_DI3.PDOS.digitalInput_12 <-> Channel 12/Input
//     PlcTask Inputs/.P1_050_DI3.PDOS.digitalInput_13 <-> Channel 13/Input
//     PlcTask Inputs/.P1_050_DI3.PDOS.digitalInput_14 <-> Channel 14/Input
//     PlcTask Inputs/.P1_050_DI3.PDOS.digitalInput_15 <-> Channel 15/Input
//     PlcTask Inputs/.P1_050_DI3.PDOS.digitalInput_16 <-> Channel 16/Input
//   Plc_Prog/Plc_Prog Instance <-> ETH/+P5=050-BC1 - PLC Cabinet/+P5=050-DO1 (EL2809)
//     PlcTask Outputs/.P1_050_DO1.PDOS.PlcToHw.digitalOutput_01 <-> Channel 1/Output
//     PlcTask Outputs/.P1_050_DO1.PDOS.PlcToHw.digitalOutput_02 <-> Channel 2/Output
//     PlcTask Outputs/.P1_050_DO1.PDOS.PlcToHw.digitalOutput_03 <-> Channel 3/Output
//     PlcTask Outputs/.P1_050_DO1.PDOS.PlcToHw.digitalOutput_04 <-> Channel 4/Output
//     PlcTask Outputs/.P1_050_DO1.PDOS.PlcToHw.digitalOutput_05 <-> Channel 5/Output
//     PlcTask Outputs/.P1_050_DO1.PDOS.PlcToHw.digitalOutput_06 <-> Channel 6/Output
//     PlcTask Outputs/.P1_050_DO1.PDOS.PlcToHw.digitalOutput_07 <-> Channel 7/Output
//     PlcTask Outputs/.P1_050_DO1.PDOS.PlcToHw.digitalOutput_08 <-> Channel 8/Output
//     PlcTask Outputs/.P1_050_DO1.PDOS.PlcToHw.digitalOutput_09 <-> Channel 9/Output
//     PlcTask Outputs/.P1_050_DO1.PDOS.PlcToHw.digitalOutput_10 <-> Channel 10/Output
//     PlcTask Outputs/.P1_050_DO1.PDOS.PlcToHw.digitalOutput_11 <-> Channel 11/Output
//     PlcTask Outputs/.P1_050_DO1.PDOS.PlcToHw.digitalOutput_12 <-> Channel 12/Output
//     PlcTask Outputs/.P1_050_DO1.PDOS.PlcToHw.digitalOutput_13 <-> Channel 13/Output
//     PlcTask Outputs/.P1_050_DO1.PDOS.PlcToHw.digitalOutput_14 <-> Channel 14/Output
//     PlcTask Outputs/.P1_050_DO1.PDOS.PlcToHw.digitalOutput_15 <-> Channel 15/Output
//     PlcTask Outputs/.P1_050_DO1.PDOS.PlcToHw.digitalOutput_16 <-> Channel 16/Output
//   Plc_Prog/Plc_Prog Instance <-> ETH/+P5=050-BC1 - PLC Cabinet/+P5=050-DO2 (EL2809)
//     PlcTask Outputs/.P1_050_DO2.PDOS.PlcToHw.digitalOutput_01 <-> Channel 1/Output
//     PlcTask Outputs/.P1_050_DO2.PDOS.PlcToHw.digitalOutput_02 <-> Channel 2/Output
//     PlcTask Outputs/.P1_050_DO2.PDOS.PlcToHw.digitalOutput_03 <-> Channel 3/Output
//     PlcTask Outputs/.P1_050_DO2.PDOS.PlcToHw.digitalOutput_04 <-> Channel 4/Output
//     PlcTask Outputs/.P1_050_DO2.PDOS.PlcToHw.digitalOutput_05 <-> Channel 5/Output
//     PlcTask Outputs/.P1_050_DO2.PDOS.PlcToHw.digitalOutput_06 <-> Channel 6/Output
//     PlcTask Outputs/.P1_050_DO2.PDOS.PlcToHw.digitalOutput_07 <-> Channel 7/Output
//     PlcTask Outputs/.P1_050_DO2.PDOS.PlcToHw.digitalOutput_08 <-> Channel 8/Output
//     PlcTask Outputs/.P1_050_DO2.PDOS.PlcToHw.digitalOutput_09 <-> Channel 9/Output
//     PlcTask Outputs/.P1_050_DO2.PDOS.PlcToHw.digitalOutput_10 <-> Channel 10/Output
//     PlcTask Outputs/.P1_050_DO2.PDOS.PlcToHw.digitalOutput_11 <-> Channel 11/Output
//     PlcTask Outputs/.P1_050_DO2.PDOS.PlcToHw.digitalOutput_12 <-> Channel 12/Output
//     PlcTask Outputs/.P1_050_DO2.PDOS.PlcToHw.digitalOutput_13 <-> Channel 13/Output
//     PlcTask Outputs/.P1_050_DO2.PDOS.PlcToHw.digitalOutput_14 <-> Channel 14/Output
//     PlcTask Outputs/.P1_050_DO2.PDOS.PlcToHw.digitalOutput_15 <-> Channel 15/Output
//     PlcTask Outputs/.P1_050_DO2.PDOS.PlcToHw.digitalOutput_16 <-> Channel 16/Output
//   Plc_Prog/Plc_Prog Instance <-> ETH/+P5=050-BC1 - PLC Cabinet/+P5=050-DO3 (EL2809)
//     PlcTask Outputs/.P1_050_DO3.PDOS.PlcToHw.digitalOutput_01 <-> Channel 1/Output
//     PlcTask Outputs/.P1_050_DO3.PDOS.PlcToHw.digitalOutput_02 <-> Channel 2/Output
//     PlcTask Outputs/.P1_050_DO3.PDOS.PlcToHw.digitalOutput_03 <-> Channel 3/Output
//     PlcTask Outputs/.P1_050_DO3.PDOS.PlcToHw.digitalOutput_04 <-> Channel 4/Output
//     PlcTask Outputs/.P1_050_DO3.PDOS.PlcToHw.digitalOutput_05 <-> Channel 5/Output
//     PlcTask Outputs/.P1_050_DO3.PDOS.PlcToHw.digitalOutput_06 <-> Channel 6/Output
//     PlcTask Outputs/.P1_050_DO3.PDOS.PlcToHw.digitalOutput_07 <-> Channel 7/Output
//     PlcTask Outputs/.P1_050_DO3.PDOS.PlcToHw.digitalOutput_08 <-> Channel 8/Output
//     PlcTask Outputs/.P1_050_DO3.PDOS.PlcToHw.digitalOutput_09 <-> Channel 9/Output
//     PlcTask Outputs/.P1_050_DO3.PDOS.PlcToHw.digitalOutput_10 <-> Channel 10/Output
//     PlcTask Outputs/.P1_050_DO3.PDOS.PlcToHw.digitalOutput_11 <-> Channel 11/Output
//     PlcTask Outputs/.P1_050_DO3.PDOS.PlcToHw.digitalOutput_12 <-> Channel 12/Output
//     PlcTask Outputs/.P1_050_DO3.PDOS.PlcToHw.digitalOutput_13 <-> Channel 13/Output
//     PlcTask Outputs/.P1_050_DO3.PDOS.PlcToHw.digitalOutput_14 <-> Channel 14/Output
//     PlcTask Outputs/.P1_050_DO3.PDOS.PlcToHw.digitalOutput_15 <-> Channel 15/Output
//     PlcTask Outputs/.P1_050_DO3.PDOS.PlcToHw.digitalOutput_16 <-> Channel 16/Output
//   Plc_Prog/Plc_Prog Instance <-> ETH/+P5=050-BC1 - PLC Cabinet/+P5=050-SP1 (EL6910)
//     PlcTask Inputs/.P1_050_SP1.PDOS.HwToPLC.EStop1Diag <-> Function Block Info Data/TwinSafeGroup1.Network1.FBEstop1 Info Data/Diag
//     PlcTask Inputs/.P1_050_SP1.PDOS.HwToPLC.EStop2Diag <-> Function Block Info Data/TwinSafeGroup1.Network1.FBEstop2 Info Data/Diag
//     PlcTask Inputs/.P1_050_SP1.PDOS.HwToPLC.EStop3Diag <-> Function Block Info Data/TwinSafeGroup1.Network1.FBEstop3 Info Data/Diag
//     PlcTask Inputs/.P1_050_SP1.PDOS.HwToPLC.EStop1State <-> Function Block Info Data/TwinSafeGroup1.Network1.FBEstop1 Info Data/State
//     PlcTask Inputs/.P1_050_SP1.PDOS.HwToPLC.EStop2State <-> Function Block Info Data/TwinSafeGroup1.Network1.FBEstop2 Info Data/State
//     PlcTask Inputs/.P1_050_SP1.PDOS.HwToPLC.EStop3State <-> Function Block Info Data/TwinSafeGroup1.Network1.FBEstop3 Info Data/State
//     PlcTask Outputs/.P1_050_SP1.PDOS.PlcToHw.ErrorAcknowledgement <-> StandardOutputs/TwinSafeGroup1.ErrorAcknowledgement_1
//     PlcTask Outputs/.P1_050_SP1.PDOS.PlcToHw.Run <-> StandardOutputs/TwinSafeGroup1.Run_2
//     PlcTask Outputs/.P1_050_SP1.PDOS.PlcToHw.safetyReset <-> StandardOutputs/TwinSafeGroup1.SafetyReset_6
//   Plc_Prog/Plc_Prog Instance <-> ETH/+P5=050-BC2 - PLC Cabinet/+P5=050-AI (EL3052)
//     PlcTask Inputs/.P1_050_AI1.PDOS.HwToPLC.Channel1/Status/Error <-> AI Standard Channel 1/Status/TxPDO Toggle
//     PlcTask Inputs/.P1_050_AI1.PDOS.HwToPLC.Channel1/Status/Limit1 <-> AI Standard Channel 1/Status/Error
//     PlcTask Inputs/.P1_050_AI1.PDOS.HwToPLC.Channel1/Status/Limit2 <-> AI Standard Channel 1/Status/TxPDO State
//     PlcTask Inputs/.P1_050_AI1.PDOS.HwToPLC.Channel1/Status/Overrange <-> AI Standard Channel 1/Status/Overrange
//     PlcTask Inputs/.P1_050_AI1.PDOS.HwToPLC.Channel2/Status/Overrange <-> AI Standard Channel 2/Status/Overrange
//     PlcTask Inputs/.P1_050_AI1.PDOS.HwToPLC.Channel1/Status/Underrange <-> AI Standard Channel 1/Status/Underrange
//     PlcTask Inputs/.P1_050_AI1.PDOS.HwToPLC.Channel2/Status/Underrange <-> AI Standard Channel 2/Status/Underrange
//     PlcTask Inputs/.P1_050_AI1.PDOS.HwToPLC.Channel1/Value <-> AI Standard Channel 1/Value
//     PlcTask Inputs/.P1_050_AI1.PDOS.HwToPLC.Channel2/Value <-> AI Standard Channel 2/Value
//     PlcTask Inputs/.P1_050_AI1.PDOS.HwToPLC.Channel2/Status/Error <-> AI Standard Channel 2/Status/Error
//     PlcTask Inputs/.P1_050_AI1.PDOS.HwToPLC.Channel2/Status/TxPDOState <-> AI Standard Channel 2/Status/TxPDO State
//     PlcTask Inputs/.P1_050_AI1.PDOS.HwToPLC.Channel2/Status/TxPDOToggle <-> AI Standard Channel 2/Status/TxPDO Toggle
//   Plc_Prog/Plc_Prog Instance <-> ETH/+P5=050-BC2 - PLC Cabinet/+P5=050-AI2 (EL3152)
//     PlcTask Inputs/.P1_050_AI2.PDOS.HwToPLC.Channel1/Status/Error <-> AI Standard Channel 1/Status/Error
//     PlcTask Inputs/.P1_050_AI2.PDOS.HwToPLC.Channel2/Status/Error <-> AI Standard Channel 2/Status/Error
//     PlcTask Inputs/.P1_050_AI2.PDOS.HwToPLC.Channel1/Status/Overrange <-> AI Standard Channel 1/Status/Overrange
//     PlcTask Inputs/.P1_050_AI2.PDOS.HwToPLC.Channel2/Status/Overrange <-> AI Standard Channel 2/Status/Overrange
//     PlcTask Inputs/.P1_050_AI2.PDOS.HwToPLC.Channel1/Status/TxPDOState <-> AI Standard Channel 1/Status/TxPDO State
//     PlcTask Inputs/.P1_050_AI2.PDOS.HwToPLC.Channel2/Status/TxPDOState <-> AI Standard Channel 2/Status/TxPDO State
//     PlcTask Inputs/.P1_050_AI2.PDOS.HwToPLC.Channel1/Status/TxPDOToggle <-> AI Standard Channel 1/Status/TxPDO Toggle
//     PlcTask Inputs/.P1_050_AI2.PDOS.HwToPLC.Channel2/Status/TxPDOToggle <-> AI Standard Channel 2/Status/TxPDO Toggle
//     PlcTask Inputs/.P1_050_AI2.PDOS.HwToPLC.Channel1/Status/Underrange <-> AI Standard Channel 1/Status/Underrange
//     PlcTask Inputs/.P1_050_AI2.PDOS.HwToPLC.Channel2/Status/Underrange <-> AI Standard Channel 2/Status/Underrange
//     PlcTask Inputs/.P1_050_AI2.PDOS.HwToPLC.Channel1/Value <-> AI Standard Channel 1/Value
//     PlcTask Inputs/.P1_050_AI2.PDOS.HwToPLC.Channel2/Value <-> AI Standard Channel 2/Value
//   Plc_Prog/Plc_Prog Instance <-> ETH/+P5=050-BC2 - PLC Cabinet/+P5=050-AI3 (EL3052)
//     PlcTask Inputs/.P1_050_AI3.PDOS.HwToPLC.Channel1/Status/Error <-> AI Standard Channel 1/Status/Error
//     PlcTask Inputs/.P1_050_AI3.PDOS.HwToPLC.Channel2/Status/Error <-> AI Standard Channel 2/Status/Error
//     PlcTask Inputs/.P1_050_AI3.PDOS.HwToPLC.Channel1/Status/Overrange <-> AI Standard Channel 1/Status/Overrange
//     PlcTask Inputs/.P1_050_AI3.PDOS.HwToPLC.Channel2/Status/Overrange <-> AI Standard Channel 2/Status/Overrange
//     PlcTask Inputs/.P1_050_AI3.PDOS.HwToPLC.Channel1/Status/TxPDOState <-> AI Standard Channel 1/Status/TxPDO State
//     PlcTask Inputs/.P1_050_AI3.PDOS.HwToPLC.Channel2/Status/TxPDOState <-> AI Standard Channel 2/Status/TxPDO State
//     PlcTask Inputs/.P1_050_AI3.PDOS.HwToPLC.Channel1/Status/TxPDOToggle <-> AI Standard Channel 1/Status/TxPDO Toggle
//     PlcTask Inputs/.P1_050_AI3.PDOS.HwToPLC.Channel2/Status/TxPDOToggle <-> AI Standard Channel 2/Status/TxPDO Toggle
//     PlcTask Inputs/.P1_050_AI3.PDOS.HwToPLC.Channel1/Status/Underrange <-> AI Standard Channel 1/Status/Underrange
//     PlcTask Inputs/.P1_050_AI3.PDOS.HwToPLC.Channel2/Status/Underrange <-> AI Standard Channel 2/Status/Underrange
//     PlcTask Inputs/.P1_050_AI3.PDOS.HwToPLC.Channel1/Value <-> AI Standard Channel 1/Value
//     PlcTask Inputs/.P1_050_AI3.PDOS.HwToPLC.Channel2/Value <-> AI Standard Channel 2/Value
//   Plc_Prog/Plc_Prog Instance <-> ETH/+P5=050-BC2 - PLC Cabinet/+P5=050-AI4 (EL3052)
//     PlcTask Inputs/.P1_050_AI4.PDOS.HwToPLC.Channel1/Status/Error <-> AI Standard Channel 1/Status/Error
//     PlcTask Inputs/.P1_050_AI4.PDOS.HwToPLC.Channel2/Status/Error <-> AI Standard Channel 2/Status/Error
//     PlcTask Inputs/.P1_050_AI4.PDOS.HwToPLC.Channel1/Status/Overrange <-> AI Standard Channel 1/Status/Overrange
//     PlcTask Inputs/.P1_050_AI4.PDOS.HwToPLC.Channel2/Status/Overrange <-> AI Standard Channel 2/Status/Overrange
//     PlcTask Inputs/.P1_050_AI4.PDOS.HwToPLC.Channel1/Status/TxPDOState <-> AI Standard Channel 1/Status/TxPDO State
//     PlcTask Inputs/.P1_050_AI4.PDOS.HwToPLC.Channel2/Status/TxPDOState <-> AI Standard Channel 2/Status/TxPDO State
//     PlcTask Inputs/.P1_050_AI4.PDOS.HwToPLC.Channel1/Status/TxPDOToggle <-> AI Standard Channel 1/Status/TxPDO Toggle
//     PlcTask Inputs/.P1_050_AI4.PDOS.HwToPLC.Channel2/Status/TxPDOToggle <-> AI Standard Channel 2/Status/TxPDO Toggle
//     PlcTask Inputs/.P1_050_AI4.PDOS.HwToPLC.Channel1/Status/Underrange <-> AI Standard Channel 1/Status/Underrange
//     PlcTask Inputs/.P1_050_AI4.PDOS.HwToPLC.Channel2/Status/Underrange <-> AI Standard Channel 2/Status/Underrange
//     PlcTask Inputs/.P1_050_AI4.PDOS.HwToPLC.Channel1/Value <-> AI Standard Channel 1/Value
//     PlcTask Inputs/.P1_050_AI4.PDOS.HwToPLC.Channel2/Value <-> AI Standard Channel 2/Value
//   Plc_Prog/Plc_Prog Instance <-> ETH/+P9=050-BC1 - Vaccum PLC Cabinet/+P9=050-AI1 (EL3054)
//     PlcTask Inputs/.P9_050_AI1.PDOS.HwToPLC.Channel1/Status/Error <-> AI Standard Channel 1/Status/Error
//     PlcTask Inputs/.P9_050_AI1.PDOS.HwToPLC.Channel2/Status/Error <-> AI Standard Channel 2/Status/Error
//     PlcTask Inputs/.P9_050_AI1.PDOS.HwToPLC.Channel1/Status/Overrange <-> AI Standard Channel 1/Status/Overrange
//     PlcTask Inputs/.P9_050_AI1.PDOS.HwToPLC.Channel2/Status/Overrange <-> AI Standard Channel 2/Status/Overrange
//     PlcTask Inputs/.P9_050_AI1.PDOS.HwToPLC.Channel1/Status/TxPDOState <-> AI Standard Channel 1/Status/TxPDO State
//     PlcTask Inputs/.P9_050_AI1.PDOS.HwToPLC.Channel2/Status/TxPDOState <-> AI Standard Channel 2/Status/TxPDO State
//     PlcTask Inputs/.P9_050_AI1.PDOS.HwToPLC.Channel1/Status/TxPDOToggle <-> AI Standard Channel 1/Status/TxPDO Toggle
//     PlcTask Inputs/.P9_050_AI1.PDOS.HwToPLC.Channel2/Status/TxPDOToggle <-> AI Standard Channel 2/Status/TxPDO Toggle
//     PlcTask Inputs/.P9_050_AI1.PDOS.HwToPLC.Channel1/Status/Underrange <-> AI Standard Channel 1/Status/Underrange
//     PlcTask Inputs/.P9_050_AI1.PDOS.HwToPLC.Channel2/Status/Underrange <-> AI Standard Channel 2/Status/Underrange
//     PlcTask Inputs/.P9_050_AI1.PDOS.HwToPLC.Channel1/Value <-> AI Standard Channel 1/Value
//     PlcTask Inputs/.P9_050_AI1.PDOS.HwToPLC.Channel2/Value <-> AI Standard Channel 2/Value
//   Plc_Prog/Plc_Prog Instance <-> ETH/+P9=050-BC1 - Vaccum PLC Cabinet/+P9=050-DI1 (EL1809)
//     PlcTask Inputs/.P9_050_DI1.PDOS.digitalInput_01 <-> Channel 1/Input
//     PlcTask Inputs/.P9_050_DI1.PDOS.digitalInput_02 <-> Channel 2/Input
//     PlcTask Inputs/.P9_050_DI1.PDOS.digitalInput_03 <-> Channel 3/Input
//     PlcTask Inputs/.P9_050_DI1.PDOS.digitalInput_04 <-> Channel 4/Input
//     PlcTask Inputs/.P9_050_DI1.PDOS.digitalInput_05 <-> Channel 5/Input
//     PlcTask Inputs/.P9_050_DI1.PDOS.digitalInput_06 <-> Channel 6/Input
//     PlcTask Inputs/.P9_050_DI1.PDOS.digitalInput_07 <-> Channel 7/Input
//     PlcTask Inputs/.P9_050_DI1.PDOS.digitalInput_08 <-> Channel 8/Input
//     PlcTask Inputs/.P9_050_DI1.PDOS.digitalInput_09 <-> Channel 9/Input
//     PlcTask Inputs/.P9_050_DI1.PDOS.digitalInput_10 <-> Channel 10/Input
//     PlcTask Inputs/.P9_050_DI1.PDOS.digitalInput_11 <-> Channel 11/Input
//     PlcTask Inputs/.P9_050_DI1.PDOS.digitalInput_12 <-> Channel 12/Input
//     PlcTask Inputs/.P9_050_DI1.PDOS.digitalInput_13 <-> Channel 13/Input
//     PlcTask Inputs/.P9_050_DI1.PDOS.digitalInput_14 <-> Channel 14/Input
//     PlcTask Inputs/.P9_050_DI1.PDOS.digitalInput_15 <-> Channel 15/Input
//     PlcTask Inputs/.P9_050_DI1.PDOS.digitalInput_16 <-> Channel 16/Input
//   Plc_Prog/Plc_Prog Instance <-> ETH/+P9=050-BC1 - Vaccum PLC Cabinet/+P9=050-DI2 (EL1809)
//     PlcTask Inputs/.P9_050_DI2.PDOS.digitalInput_01 <-> Channel 1/Input
//     PlcTask Inputs/.P9_050_DI2.PDOS.digitalInput_02 <-> Channel 2/Input
//     PlcTask Inputs/.P9_050_DI2.PDOS.digitalInput_03 <-> Channel 3/Input
//     PlcTask Inputs/.P9_050_DI2.PDOS.digitalInput_04 <-> Channel 4/Input
//     PlcTask Inputs/.P9_050_DI2.PDOS.digitalInput_05 <-> Channel 5/Input
//     PlcTask Inputs/.P9_050_DI2.PDOS.digitalInput_06 <-> Channel 6/Input
//     PlcTask Inputs/.P9_050_DI2.PDOS.digitalInput_07 <-> Channel 7/Input
//     PlcTask Inputs/.P9_050_DI2.PDOS.digitalInput_08 <-> Channel 8/Input
//     PlcTask Inputs/.P9_050_DI2.PDOS.digitalInput_09 <-> Channel 9/Input
//     PlcTask Inputs/.P9_050_DI2.PDOS.digitalInput_10 <-> Channel 10/Input
//     PlcTask Inputs/.P9_050_DI2.PDOS.digitalInput_11 <-> Channel 11/Input
//     PlcTask Inputs/.P9_050_DI2.PDOS.digitalInput_12 <-> Channel 12/Input
//     PlcTask Inputs/.P9_050_DI2.PDOS.digitalInput_13 <-> Channel 13/Input
//     PlcTask Inputs/.P9_050_DI2.PDOS.digitalInput_14 <-> Channel 14/Input
//     PlcTask Inputs/.P9_050_DI2.PDOS.digitalInput_15 <-> Channel 15/Input
//     PlcTask Inputs/.P9_050_DI2.PDOS.digitalInput_16 <-> Channel 16/Input
//   Plc_Prog/Plc_Prog Instance <-> ETH/+P9=050-BC1 - Vaccum PLC Cabinet/+P9=050-DI3 (EL1809)
//     PlcTask Inputs/.P9_050_DI3.PDOS.digitalInput_01 <-> Channel 1/Input
//     PlcTask Inputs/.P9_050_DI3.PDOS.digitalInput_02 <-> Channel 2/Input
//     PlcTask Inputs/.P9_050_DI3.PDOS.digitalInput_03 <-> Channel 3/Input
//     PlcTask Inputs/.P9_050_DI3.PDOS.digitalInput_04 <-> Channel 4/Input
//     PlcTask Inputs/.P9_050_DI3.PDOS.digitalInput_05 <-> Channel 5/Input
//     PlcTask Inputs/.P9_050_DI3.PDOS.digitalInput_06 <-> Channel 6/Input
//     PlcTask Inputs/.P9_050_DI3.PDOS.digitalInput_07 <-> Channel 7/Input
//     PlcTask Inputs/.P9_050_DI3.PDOS.digitalInput_08 <-> Channel 8/Input
//     PlcTask Inputs/.P9_050_DI3.PDOS.digitalInput_09 <-> Channel 9/Input
//     PlcTask Inputs/.P9_050_DI3.PDOS.digitalInput_10 <-> Channel 10/Input
//     PlcTask Inputs/.P9_050_DI3.PDOS.digitalInput_11 <-> Channel 11/Input
//     PlcTask Inputs/.P9_050_DI3.PDOS.digitalInput_12 <-> Channel 12/Input
//     PlcTask Inputs/.P9_050_DI3.PDOS.digitalInput_13 <-> Channel 13/Input
//     PlcTask Inputs/.P9_050_DI3.PDOS.digitalInput_14 <-> Channel 14/Input
//     PlcTask Inputs/.P9_050_DI3.PDOS.digitalInput_15 <-> Channel 15/Input
//     PlcTask Inputs/.P9_050_DI3.PDOS.digitalInput_16 <-> Channel 16/Input
//   Plc_Prog/Plc_Prog Instance <-> ETH/+P9=050-BC1 - Vaccum PLC Cabinet/+P9=050-DO1 (EL2809)
//     PlcTask Outputs/.P9_050_DO1.PDOS.PlcToHw.digitalOutput_01 <-> Channel 1/Output
//     PlcTask Outputs/.P9_050_DO1.PDOS.PlcToHw.digitalOutput_02 <-> Channel 2/Output
//     PlcTask Outputs/.P9_050_DO1.PDOS.PlcToHw.digitalOutput_03 <-> Channel 3/Output
//     PlcTask Outputs/.P9_050_DO1.PDOS.PlcToHw.digitalOutput_04 <-> Channel 4/Output
//     PlcTask Outputs/.P9_050_DO1.PDOS.PlcToHw.digitalOutput_05 <-> Channel 5/Output
//     PlcTask Outputs/.P9_050_DO1.PDOS.PlcToHw.digitalOutput_06 <-> Channel 6/Output
//     PlcTask Outputs/.P9_050_DO1.PDOS.PlcToHw.digitalOutput_07 <-> Channel 7/Output
//     PlcTask Outputs/.P9_050_DO1.PDOS.PlcToHw.digitalOutput_08 <-> Channel 8/Output
//     PlcTask Outputs/.P9_050_DO1.PDOS.PlcToHw.digitalOutput_09 <-> Channel 9/Output
//     PlcTask Outputs/.P9_050_DO1.PDOS.PlcToHw.digitalOutput_10 <-> Channel 10/Output
//     PlcTask Outputs/.P9_050_DO1.PDOS.PlcToHw.digitalOutput_11 <-> Channel 11/Output
//     PlcTask Outputs/.P9_050_DO1.PDOS.PlcToHw.digitalOutput_12 <-> Channel 12/Output
//     PlcTask Outputs/.P9_050_DO1.PDOS.PlcToHw.digitalOutput_13 <-> Channel 13/Output
//     PlcTask Outputs/.P9_050_DO1.PDOS.PlcToHw.digitalOutput_14 <-> Channel 14/Output
//     PlcTask Outputs/.P9_050_DO1.PDOS.PlcToHw.digitalOutput_15 <-> Channel 15/Output
//     PlcTask Outputs/.P9_050_DO1.PDOS.PlcToHw.digitalOutput_16 <-> Channel 16/Output
//   Plc_Prog/Plc_Prog Instance <-> ETH/+P9=050-BC1 - Vaccum PLC Cabinet/+P9=050-DO2 (EL2809)
//     PlcTask Outputs/.P9_050_DO2.PDOS.PlcToHw.digitalOutput_01 <-> Channel 1/Output
//     PlcTask Outputs/.P9_050_DO2.PDOS.PlcToHw.digitalOutput_02 <-> Channel 2/Output
//     PlcTask Outputs/.P9_050_DO2.PDOS.PlcToHw.digitalOutput_03 <-> Channel 3/Output
//     PlcTask Outputs/.P9_050_DO2.PDOS.PlcToHw.digitalOutput_04 <-> Channel 4/Output
//     PlcTask Outputs/.P9_050_DO2.PDOS.PlcToHw.digitalOutput_05 <-> Channel 5/Output
//     PlcTask Outputs/.P9_050_DO2.PDOS.PlcToHw.digitalOutput_06 <-> Channel 6/Output
//     PlcTask Outputs/.P9_050_DO2.PDOS.PlcToHw.digitalOutput_07 <-> Channel 7/Output
//     PlcTask Outputs/.P9_050_DO2.PDOS.PlcToHw.digitalOutput_08 <-> Channel 8/Output
//     PlcTask Outputs/.P9_050_DO2.PDOS.PlcToHw.digitalOutput_09 <-> Channel 9/Output
//     PlcTask Outputs/.P9_050_DO2.PDOS.PlcToHw.digitalOutput_10 <-> Channel 10/Output
//     PlcTask Outputs/.P9_050_DO2.PDOS.PlcToHw.digitalOutput_11 <-> Channel 11/Output
//     PlcTask Outputs/.P9_050_DO2.PDOS.PlcToHw.digitalOutput_12 <-> Channel 12/Output
//     PlcTask Outputs/.P9_050_DO2.PDOS.PlcToHw.digitalOutput_13 <-> Channel 13/Output
//     PlcTask Outputs/.P9_050_DO2.PDOS.PlcToHw.digitalOutput_14 <-> Channel 14/Output
//     PlcTask Outputs/.P9_050_DO2.PDOS.PlcToHw.digitalOutput_15 <-> Channel 15/Output
//     PlcTask Outputs/.P9_050_DO2.PDOS.PlcToHw.digitalOutput_16 <-> Channel 16/Output
//   Plc_Prog/Plc_Prog Instance <-> ETH/+P9=050-BC1 - Vaccum PLC Cabinet/+P9=050-DO3 (EL2809)
//     PlcTask Outputs/.P9_050_DO3.PDOS.PlcToHw.digitalOutput_01 <-> Channel 1/Output
//     PlcTask Outputs/.P9_050_DO3.PDOS.PlcToHw.digitalOutput_02 <-> Channel 2/Output
//     PlcTask Outputs/.P9_050_DO3.PDOS.PlcToHw.digitalOutput_06 <-> Channel 6/Output
//     PlcTask Outputs/.P9_050_DO3.PDOS.PlcToHw.digitalOutput_07 <-> Channel 7/Output
//     PlcTask Outputs/.P9_050_DO3.PDOS.PlcToHw.digitalOutput_08 <-> Channel 8/Output
//     PlcTask Outputs/.P9_050_DO3.PDOS.PlcToHw.digitalOutput_09 <-> Channel 9/Output
//     PlcTask Outputs/.P9_050_DO3.PDOS.PlcToHw.digitalOutput_10 <-> Channel 10/Output
//     PlcTask Outputs/.P9_050_DO3.PDOS.PlcToHw.digitalOutput_11 <-> Channel 11/Output
//     PlcTask Outputs/.P9_050_DO3.PDOS.PlcToHw.digitalOutput_12 <-> Channel 12/Output
//     PlcTask Outputs/.P9_050_DO3.PDOS.PlcToHw.digitalOutput_13 <-> Channel 13/Output
//     PlcTask Outputs/.P9_050_DO3.PDOS.PlcToHw.digitalOutput_14 <-> Channel 14/Output
//     PlcTask Outputs/.P9_050_DO3.PDOS.PlcToHw.digitalOutput_15 <-> Channel 15/Output
//     PlcTask Outputs/.P9_050_DO3.PDOS.PlcToHw.digitalOutput_16 <-> Channel 16/Output
//     PlcTask Outputs/.P9_050_DO3.PDOS.PlcToHw.digitalOutput_03 <-> Channel 3/Libera Safety Vacuo
//     PlcTask Outputs/.P9_050_DO3.PDOS.PlcToHw.digitalOutput_04 <-> Channel 4/Selagem do vacuo
//     PlcTask Outputs/.P9_050_DO3.PDOS.PlcToHw.digitalOutput_05 <-> Channel 5/Separador Baixo Vacuo
//   Plc_Prog/Plc_Prog Instance <-> ETH/+P9=050-BC1 - Vaccum PLC Cabinet/Term 101 (EL3052)
//     PlcTask Inputs/.P9_050_AI2.PDOS.HwToPLC.Channel1/Status/Overrange <-> AI Standard Channel 1/Status/Overrange
//     PlcTask Inputs/.P9_050_AI2.PDOS.HwToPLC.Channel1/Status/Underrange <-> AI Standard Channel 1/Status/Underrange
//     PlcTask Inputs/.P9_050_AI2.PDOS.HwToPLC.Channel1/Value <-> AI Standard Channel 1/Value
//     PlcTask Inputs/.P9_050_AI2.PDOS.HwToPLC.Channel2/Value <-> AI Standard Channel 2/Value
//     PlcTask Inputs/.P9_050_AI2.PDOS.HwToPLC.Channel2/Status/Overrange <-> AI Standard Channel 2/Status/Underrange
//   Plc_Prog/Plc_Prog Instance <-> ETH/+P9=050-BC1 - Vaccum PLC Cabinet/Term 102 (EL4004)
//     PlcTask Outputs/.P9_050_AQ1.PDOS.HwToPLC.Channel1 <-> AO Outputs Channel 1/Analog output
//     PlcTask Outputs/.P9_050_AQ1.PDOS.HwToPLC.Channel2 <-> AO Outputs Channel 2/Analog output
//     PlcTask Outputs/.P9_050_AQ1.PDOS.HwToPLC.Channel3 <-> AO Outputs Channel 3/Analog output
//     PlcTask Outputs/.P9_050_AQ1.PDOS.HwToPLC.Channel4 <-> AO Outputs Channel 4/Analog output

CONFIGURATION Plc_Prog
    RESOURCE PLC ON TwinCAT3
        TASK PlcTask(INTERVAL := T#5ms, PRIORITY := 20);
        PROGRAM MAIN WITH PlcTask : MAIN;
    END_RESOURCE
END_CONFIGURATION

// ---- Function Blocks/DELTA - MS300/C2000_DEV_CONFIG.TcDUT
TYPE C2000_DEV_CONFIG :
    STRUCT
        // Setpoint scaling
        speedSetpointInputLow        : REAL := 0.0;   // Minimum input value for setpoint		
        speedSetpointInputHigh       : REAL := 100.0; // Maximum input value for setpoint
        speedSetpointOutputLow       : REAL := 0.0; // Minimum output value for setpoint
        speedSetpointOutputHigh      : REAL := 6000.0; // Maximum output value for setpoint
		
        torqueSetpointInputLow        : REAL := 0.0;   // Minimum input value for setpoint
        torqueSetpointInputHigh       : REAL := 100.0; // Maximum input value for setpoint
        torqueSetpointOutputLow       : REAL := 0.0; // Minimum output value for setpoint				
        torqueSetpointOutputHigh      : REAL := 1000; // Maximum output value for setpoint
		
		torqueLimiterEnabled			: BOOL := FALSE;
		torqueDif						: REAL := 0.0;

        // Motor speed scaling
        MotorSpeedInputLow      : REAL := 0.0;    // Minimum input value for motor speed		
        MotorSpeedInputHigh     : REAL := 6000.0; // Maximum input value for motor speed
        MotorSpeedOutputLow     : REAL := 0.0;    // Minimum output value for motor speed		
        MotorSpeedOutputHigh    : REAL := 100.0;  // Maximum output value for motor speed
		
		
        // Motor speed MPM scaling
        MotorSpeedMPMOutputLow     : REAL := 0.0;    // Minimum output value for motor speed		
        MotorSpeedMPMOutputHigh    : REAL := 600.0;  // Maximum output value for motor speed
		

        // Output current scaling
        OutputCurrentInputLow   : REAL	:= 0; 		// Minimum input value for output current		
        OutputCurrentInputHigh  : REAL	:= 10000.0; // Maximum input value for output current
        OutputCurrentOutputLow  : REAL 	:= 0.0;		// Minimum output value for output current		
        OutputCurrentOutputHigh : REAL	:= 100.0; 	// Maximum output value for output current

        // Output torque scaling
        OutputTorqueInputLow    : REAL := -1500.0;     // Minimum input value for output torque		
        OutputTorqueInputHigh   : REAL := 1500.0; // Maximum input value for output torque
        OutputTorqueOutputLow   : REAL := -150.0;     // Minimum output value for output torque		
        OutputTorqueOutputHigh  : REAL := 150.0;   // Maximum output value for output torque

        // Current scaling
        currentInputHigh        : REAL := 10000; // Maximum input value for current
        currentaviInputLow      : REAL := 0;     // Minimum input value for current
        currentOutputHigh       : REAL := 100.0; // Maximum output value for current
        currentOutputLow        : REAL := 0.0;   // Minimum output value for current

        // Operation mode
        operationMode           : E_C2000_ModeOfOperation := 2; // 0 - Reserved / 1 - Profile Position Mode / 2 - Velocity Mode / 3 - Reserved / 4 - Profile Torque Mode

    END_STRUCT
END_TYPE

// ---- Function Blocks/DELTA - MS300/C2000_DIGITAL_INPUTS.TcDUT
TYPE C2000_DIGITAL_INPUTS :
STRUCT
		
	MI1					: BOOL; (*Drive digital input - Term M1*)
	MI2					: BOOL; (*Drive digital input - Term M2*)
	MI3					: BOOL; (*Drive digital input - Term M3*)
	MI4					: BOOL; (*Drive digital input - Term M4*)
	MI5					: BOOL; (*Drive digital input - Term M5*)
	MI6					: BOOL; (*Drive digital input - Term M6*)
	MI7					: BOOL; (*Drive digital input - Term M7*)
	MI8					: BOOL; (*Drive digital input - Term M8*)
		
END_STRUCT
END_TYPE

// ---- Function Blocks/DELTA - MS300/C2000_PDOS.TcDUT
TYPE C2000_PDOS :
STRUCT
	
	DrvToPLC : C2000_DRVTOPLC_PDOS;
	PlcToDrv : C2000_PLCTODRV_PDOS;		

END_STRUCT
END_TYPE

// ---- Function Blocks/DELTA - MS300/E_C2000_ModeOfOperation.TcDUT
{attribute 'qualified_only'}
{attribute 'strict'}
TYPE E_C2000_ModeOfOperation :
(
    Reserved_0                      := 0,  // Reserved
    ProfilePositionMode             := 1,  // Profile Position Mode
    VelocityMode                    := 2,  // Velocity Mode
    Reserved_3                      := 3,  // Reserved
    ProfileTorqueMode               := 4,  // Profile Torque Mode
    Reserved_5                      := 5,  // Reserved
    HomingMode                      := 6,  // Homing Mode
    Reserved_7                      := 7,  // Reserved (not listed but keeps alignment)
    CyclicSynchronousPositionMode   := 8,  // Cyclic Synchronous Position Mode
    Reserved_9                      := 9,  // Reserved
    CyclicSynchronousTorqueMode     := 10  // Cyclic Synchronous Torque Mode
);
END_TYPE

// ---- Function Blocks/IOs/Beckhoff/EL1809 - Digital Inputs/DataTypes/EL1809_DEV_CONFIG.TcDUT
TYPE EL1809_DEV_CONFIG :
    STRUCT
       
		enableForce	: BOOL;
		forceDigitalInput_00 : BOOL;
		forceDigitalInput_01 : BOOL;
		forceDigitalInput_02 : BOOL;
		forceDigitalInput_03 : BOOL;
		forceDigitalInput_04 : BOOL;
		forceDigitalInput_05 : BOOL;
		forceDigitalInput_06 : BOOL;
		forceDigitalInput_07 : BOOL;
		forceDigitalInput_08 : BOOL;
		forceDigitalInput_09 : BOOL;
		forceDigitalInput_10 : BOOL;
		forceDigitalInput_11 : BOOL;
		forceDigitalInput_12 : BOOL;
		forceDigitalInput_13 : BOOL;
		forceDigitalInput_14 : BOOL;
		forceDigitalInput_15 : BOOL;


    END_STRUCT
END_TYPE

// ---- Function Blocks/IOs/Beckhoff/EL1809 - Digital Inputs/DataTypes/EL1809_PDOS.TcDUT
TYPE EL1809_PDOS :
	STRUCT
		
		HwToPLC : EL1809_HWTOPLC_PDOS;
		
	END_STRUCT
END_TYPE

// ---- Function Blocks/IOs/Beckhoff/EL3052 - Ai 2 x 4-20MA - 12bit/DataTypes/EL3052_CHANNEL.TcDUT
TYPE EL3052_CHANNEL :
	STRUCT
		
	
	Status 	AT %I* : EL3052_DEV_STATUS;
	Value 	AT %I* : INT;
	
	
	END_STRUCT
END_TYPE

// ---- Function Blocks/IOs/Beckhoff/EL3052 - Ai 2 x 4-20MA - 12bit/DataTypes/EL3052_PDOS.TcDUT
TYPE EL3052_PDOS :
	STRUCT
		
		HwToPLC : EL3052_HWTOPLC_PDOS;
		
	END_STRUCT
END_TYPE

// ---- Function Blocks/IOs/Beckhoff/EL2809 - Digital Outputs/DataTypes/EL2809_PDOS.TcDUT
TYPE EL2809_PDOS :
	STRUCT
		
		PlcToHw : EL2809_PLCTOHW_PDOS;
		
	END_STRUCT
END_TYPE

// ---- Function Blocks/IOs/Beckhoff/EL3152 - Ai 2 x 4-20MA - 16bit/DataTypes/EL3152_HWTOPLC_PDOS.TcDUT
TYPE EL3152_HWTOPLC_PDOS :
	STRUCT
		
	
	Channel1 	AT %I* : EL3152_CHANNEL;
	Channel2 	AT %I* : EL3152_CHANNEL;



	END_STRUCT
END_TYPE

// ---- Function Blocks/IOs/Beckhoff/EL3154 - Ai 4 x 4-20MA - 16bit/DataTypes/EL3154_CHANNEL.TcDUT
TYPE EL3154_CHANNEL :
	STRUCT
		
	
	Status 	AT %I* : EL3154_DEV_STATUS;
	Value 	AT %I* : INT;
	
	
	END_STRUCT
END_TYPE

// ---- Function Blocks/IOs/Beckhoff/EL3154 - Ai 4 x 4-20MA - 16bit/DataTypes/EL3154_HWTOPLC_PDOS.TcDUT
TYPE EL3154_HWTOPLC_PDOS :
	STRUCT
		
	
	Channel1 	AT %I* : EL3154_CHANNEL;
	Channel2 	AT %I* : EL3154_CHANNEL;
	Channel3 	AT %I* : EL3154_CHANNEL;
	Channel4 	AT %I* : EL3154_CHANNEL;



	END_STRUCT
END_TYPE

// ---- Function Blocks/IOs/Beckhoff/EL6910 - TwinSAFE PLC/EL6910_ESTOP_STATUS.TcDUT
TYPE EL6910_ESTOP_STATUS :
STRUCT
	
    estopState_RUN        : BOOL; // RUN state 
    estopState_STOP       : BOOL; // STOP state 
    estopState_SAFE       : BOOL; // SAFE state 
    estopState_ERROR      : BOOL; // ERROR state 
    estopState_RESET      : BOOL; // RESET state 
    estopState_START      : BOOL; // START state 
    estopState_DELAYOUT   : BOOL; // DELAYOUT state 
	
END_STRUCT
END_TYPE

// ---- Function Blocks/IOs/Beckhoff/EL6910 - TwinSAFE PLC/EL6910_PDOS.TcDUT
TYPE EL6910_PDOS :
STRUCT
	
	HwToPLC : EL6910_HWTOPLC_PDOS;
	PlcToHw : EL6910_PLCTOHW_PDOS;			

END_STRUCT
END_TYPE

// ---- Function Blocks/IOs/Beckhoff/EL6910 - TwinSAFE PLC/EL6910_PLCTOHW_PDOS.TcDUT
TYPE EL6910_PLCTOHW_PDOS :
	STRUCT
		
		ErrorAcknowledgement AT %Q* : BOOL;
		safetyReset AT %Q* : BOOL;
	
		Run AT %Q* : BOOL;
		
	END_STRUCT
END_TYPE

// ---- Function Blocks/PaperMachine/DataTypes/PaperMachine_TypeHmiConfig.TcDUT
TYPE PaperMachine_TypeHmiConfig :
	STRUCT
		
	
	machineRampUPRate	: REAL := 0.01;			//Forming board manual speed (Slow speed)
	machineRampDownRate	: REAL := 0.01;			//Forming board manual speed (Slow speed)
	
	machineRampUPRate2	: REAL := 0.01;			//Forming board manual speed (Slow speed)
	machineRampDownRate2	: REAL := 0.01;			//Forming board manual speed (Slow speed)
		
	
    groupSpeedDifLimLow        : REAL := -15.0;  // Min offset [%]
    groupSpeedDifLimHigh       : REAL := 15.0;  // Max offset [%]

    groupRecoverIncrement : REAL := 2.0;
	
	
	

	
	
	
	dryingSectionGroup1SteamPressureKp : REAL := 1.0;  // PID Kp for Group 1 steam pressure
	dryingSectionGroup1SteamPressureTn : REAL := 8.0;  // PID Tn for Group 1 steam pressure
	dryingSectionGroup1SteamPressureTv : REAL := 0.0;  // PID Tv for Group 1 steam pressure
	
	dryingSectionGroup2SteamPressureKp : REAL := 1.0;  // PID Kp for Group 1 steam pressure
	dryingSectionGroup2SteamPressureTn : REAL := 8.0;  // PID Tn for Group 1 steam pressure
	dryingSectionGroup2SteamPressureTv : REAL := 0.0;  // PID Tv for Group 1 steam pressure
	
